// TIA Portal V17 program export: 3 tag tables, 24 data types, 1 data blocks, 11 code blocks (in call order from the OBs), 7 instance data blocks

VAR_GLOBAL   // PLC tag table "Default tag table"
END_VAR

VAR_GLOBAL   // PLC tag table "LPMLV2022_PackTags_Constants"
END_VAR
VAR_GLOBAL CONSTANT   // user constants
   LPMLV2022_COMMAND_PARAMETER_BOOL_UPPER_LIM : UInt := 0;   // Size [0..UPPER_LIM] of structured Array of Unit/Machine Parameter information for values with BOOL data type
   LPMLV2022_COMMAND_PARAMETER_DINT_UPPER_LIM : UInt := 0;   // Size [0..UPPER_LIM] of structured Array of Unit/Machine Parameter information for values with DINT data type
   LPMLV2022_COMMAND_PARAMETER_REAL_UPPER_LIM : UInt := 0;   // Size [0..UPPER_LIM] of structured Array of Unit/Machine Parameter information for values with REAL data type
   LPMLV2022_COMMAND_PARAMETER_LREAL_UPPER_LIM : UInt := 0;   // Size [0..UPPER_LIM] of structured Array of Unit/Machine Parameter information for values with LREAL data type
   LPMLV2022_COMMAND_PARAMETER_STRING_UPPER_LIM : UInt := 0;   // Size [0..UPPER_LIM] of structured Array of Unit/Machine Parameter information for values with STRING data type
   LPMLV2022_COMMAND_RECIPE_UPPER_LIM : UInt := 0;   // Size [0..UPPER_LIM] of structured Array of Recipe Information
   LPMLV2022_COMMAND_PROCESS_VARIABLES_PARAMETER_BOOL_UPPER_LIM : UInt := 0;   // Size [0..UPPER_LIM] of structured Array of Recipe Process Variable information for values with BOOL data type
   LPMLV2022_COMMAND_PROCESS_VARIABLES_PARAMETER_DINT_UPPER_LIM : UInt := 0;   // Size [0..UPPER_LIM] of structured Array of Recipe Process Variable Information for values with DINT data type
   LPMLV2022_COMMAND_PROCESS_VARIABLES_PARAMETER_REAL_UPPER_LIM : UInt := 0;   // Size [0..UPPER_LIM] of structured Array of Recipe Process Variable information for values with REAL data type
   LPMLV2022_COMMAND_PROCESS_VARIABLES_PARAMETER_LREAL_UPPER_LIM : UInt := 0;   // Size [0..UPPER_LIM] of structured Array of Recipe Process Variable information for values with LREAL data type
   LPMLV2022_COMMAND_PROCESS_VARIABLES_PARAMETER_STRING_UPPER_LIM : UInt := 0;   // Size [0..UPPER_LIM] of structured Array of Recipe Process Variable information for values with STRING data type
   LPMLV2022_COMMAND_INGREDIENTS_PARAMETER_BOOL_UPPER_LIM : UInt := 0;   // Size [0..UPPER_LIM] of structured Array of Ingredient information for values with BOOL data type
   LPMLV2022_COMMAND_INGREDIENTS_PARAMETER_DINT_UPPER_LIM : UInt := 0;   // Size [0..UPPER_LIM] of structured Array of Ingredient Information for values with DINT data type
   LPMLV2022_COMMAND_INGREDIENTS_PARAMETER_REAL_UPPER_LIM : UInt := 0;   // Size [0..UPPER_LIM] of structured Array of Ingredient information for values with REAL data type
   LPMLV2022_COMMAND_INGREDIENTS_PARAMETER_LREAL_UPPER_LIM : UInt := 0;   // Size [0..UPPER_LIM] of structured Array of Ingredient information for values with LREAL data type
   LPMLV2022_COMMAND_INGREDIENTS_PARAMETER_STRING_UPPER_LIM : UInt := 0;   // Size [0..UPPER_LIM] of structured Array of Ingredient information for values with STRING data type
   LPMLV2022_STATUS_PARAMETER_BOOL_UPPER_LIM : UInt := 0;   // Size [0..UPPER_LIM] of structured Array of Unit/Machine Parameter information for values with BOOL data type
   LPMLV2022_STATUS_PARAMETER_DINT_UPPER_LIM : UInt := 0;   // Size [0..UPPER_LIM] of structured Array of Unit/Machine Parameter information for values with DINT data type
   LPMLV2022_STATUS_PARAMETER_REAL_UPPER_LIM : UInt := 0;   // Size [0..UPPER_LIM] of structured Array of Unit/Machine Parameter information for values with REAL data type
   LPMLV2022_STATUS_PARAMETER_LREAL_UPPER_LIM : UInt := 0;   // Size [0..UPPER_LIM] of structured Array of Unit/Machine Parameter information for values with LREAL data type
   LPMLV2022_STATUS_PARAMETER_STRING_UPPER_LIM : UInt := 0;   // Size [0..UPPER_LIM] of structured Array of Unit/Machine Parameter information for values with STRING data type
   LPMLV2022_STATUS_RECIPE_UPPER_LIM : UInt := 0;   // Size [0..UPPER_LIM] of structured Array of Recipe Information
   LPMLV2022_STATUS_PROCESS_VARIABLES_PARAMETER_BOOL_UPPER_LIM : UInt := 0;   // Size [0..UPPER_LIM] of structured Array of Recipe Process Variable information for values with BOOL data type
   LPMLV2022_STATUS_PROCESS_VARIABLES_PARAMETER_DINT_UPPER_LIM : UInt := 0;   // Size [0..UPPER_LIM] of structured Array of Recipe Process Variable Information for values with DINT data type
   LPMLV2022_STATUS_PROCESS_VARIABLES_PARAMETER_REAL_UPPER_LIM : UInt := 0;   // Size [0..UPPER_LIM] of structured Array of Recipe Process Variable information for values with REAL data type
   LPMLV2022_STATUS_PROCESS_VARIABLES_PARAMETER_LREAL_UPPER_LIM : UInt := 0;   // Size [0..UPPER_LIM] of structured Array of Recipe Process Variable information for values with LREAL data type
   LPMLV2022_STATUS_PROCESS_VARIABLES_PARAMETER_STRING_UPPER_LIM : UInt := 0;   // Size [0..UPPER_LIM] of structured Array of Recipe Process Variable information for values with STRING data type
   LPMLV2022_STATUS_INGREDIENTS_PARAMETER_BOOL_UPPER_LIM : UInt := 0;   // Size [0..UPPER_LIM] of structured Array of Ingredient information for values with BOOL data type
   LPMLV2022_STATUS_INGREDIENTS_PARAMETER_DINT_UPPER_LIM : UInt := 0;   // Size [0..UPPER_LIM] of structured Array of Ingredient Information for values with DINT data type
   LPMLV2022_STATUS_INGREDIENTS_PARAMETER_REAL_UPPER_LIM : UInt := 0;   // Size [0..UPPER_LIM] of structured Array of Ingredient information for values with REAL data type
   LPMLV2022_STATUS_INGREDIENTS_PARAMETER_LREAL_UPPER_LIM : UInt := 0;   // Size [0..UPPER_LIM] of structured Array of Ingredient information for values with LREAL data type
   LPMLV2022_STATUS_INGREDIENTS_PARAMETER_STRING_UPPER_LIM : UInt := 0;   // Size [0..UPPER_LIM] of structured Array of Ingredient information for values with STRING data type
   LPMLV2022_STATUS_STACK_LIGHT_UPPER_LIM : UInt := 0;   // Size [0..UPPER_LIM] of Indicator for the current stacklight status
   LPMLV2022_ADMIN_PARAMETER_BOOL_UPPER_LIM : UInt := 0;   // Size [0..UPPER_LIM] of structured Array of Unit/Machine Parameter information for values with BOOL data type
   LPMLV2022_ADMIN_PARAMETER_DINT_UPPER_LIM : UInt := 0;   // Size [0..UPPER_LIM] of structured Array of Unit/Machine Parameter information for values with DINT data type
   LPMLV2022_ADMIN_PARAMETER_REAL_UPPER_LIM : UInt := 0;   // Size [0..UPPER_LIM] of structured Array of Unit/Machine Parameter information for values with REAL data type
   LPMLV2022_ADMIN_PARAMETER_LREAL_UPPER_LIM : UInt := 0;   // Size [0..UPPER_LIM] of structured Array of Unit/Machine Parameter information for values with LREAL data type
   LPMLV2022_ADMIN_PARAMETER_STRING_UPPER_LIM : UInt := 0;   // Size [0..UPPER_LIM] of structured Array of Unit/Machine Parameter information for values with STRING data type
   LPMLV2022_ADMIN_ALARM_UPPER_LIM : UInt := 0;   // Size [0..UPPER_LIM] of Array for Machine Alarms
   LPMLV2022_ADMIN_ALARM_HISTORY_UPPER_LIM : UInt := 0;   // Size [0..UPPER_LIM] of Array for Machine Fault Number and Messaging History
   LPMLV2022_ADMIN_WARNING_UPPER_LIM : UInt := 0;   // Size [0..UPPER_LIM] of Machine warnings for general events that do not cause the machine to stop
   LPMLV2022_ADMIN_CUMULATIVE_TIMES_UPPER_LIM : UInt := 0;   // Size [0..UPPER_LIM] of structured Array of Timer Values
   LPMLV2022_ADMIN_NUMBER_OF_MODES_UPPER_LIM : UInt := 8;   // Size [0..UPPER_LIM] of structured Array of Mode and State Time Values for each Cumulative Time Tracker
   LPMLV2022_ADMIN_NUMBER_OF_STATES_UPPER_LIM : UInt := 17;   // Size [0..UPPER_LIM] of state Time Values for each State in each Mode
   LPMLV2022_ADMIN_PRODUCT_DATA_UPPER_LIM : UInt := 0;   // Size [0..UPPER_LIM] of structured array of Product Stream Data
END_VAR

VAR_GLOBAL   // PLC tag table "LPMLV2022_Constants"
END_VAR
VAR_GLOBAL CONSTANT   // user constants
   LPMLV2022_MODE_INVALID : DInt := 0;   // OMAC PackMLV2022 unit mode Invalid
   LPMLV2022_MODE_PRODUCTION : DInt := 1;   // OMAC PackMLV2022 unit mode Production
   LPMLV2022_MODE_MAINTENANCE : DInt := 2;   // OMAC PackMLV2022 unit mode Maintenance
   LPMLV2022_MODE_MANUAL : DInt := 3;   // OMAC PackMLV2022 unit mode Manual
   LPMLV2022_MODE_USER_01 : DInt := 4;   // OMAC PackMLV2022 user-defined unit mode 01
   LPMLV2022_MODE_USER_02 : DInt := 5;   // OMAC PackMLV2022 user-defined unit mode 02
   LPMLV2022_MODE_USER_03 : DInt := 6;   // OMAC PackMLV2022 user-defined unit mode 03
   LPMLV2022_MODE_USER_04 : DInt := 7;   // OMAC PackMLV2022 user-defined unit mode 04
   LPMLV2022_MODE_USER_05 : DInt := 8;   // OMAC PackMLV2022 user-defined unit mode 05
   LPMLV2022_MODE_USER_06 : DInt := 9;   // OMAC PackMLV2022 user-defined unit mode 06
   LPMLV2022_MODE_USER_07 : DInt := 10;   // OMAC PackMLV2022 user-defined unit mode 07
   LPMLV2022_MODE_USER_08 : DInt := 11;   // OMAC PackMLV2022 user-defined unit mode 08
   LPMLV2022_MODE_USER_09 : DInt := 12;   // OMAC PackMLV2022 user-defined unit mode 09
   LPMLV2022_MODE_USER_10 : DInt := 13;   // OMAC PackMLV2022 user-defined unit mode 10
   LPMLV2022_MODE_USER_11 : DInt := 14;   // OMAC PackMLV2022 user-defined unit mode 11
   LPMLV2022_MODE_USER_12 : DInt := 15;   // OMAC PackMLV2022 user-defined unit mode 12
   LPMLV2022_MODE_USER_13 : DInt := 16;   // OMAC PackMLV2022 user-defined unit mode 13
   LPMLV2022_MODE_USER_14 : DInt := 17;   // OMAC PackMLV2022 user-defined unit mode 14
   LPMLV2022_MODE_USER_15 : DInt := 18;   // OMAC PackMLV2022 user-defined unit mode 15
   LPMLV2022_MODE_USER_16 : DInt := 19;   // OMAC PackMLV2022 user-defined unit mode 16
   LPMLV2022_MODE_USER_17 : DInt := 20;   // OMAC PackMLV2022 user-defined unit mode 17
   LPMLV2022_MODE_USER_18 : DInt := 21;   // OMAC PackMLV2022 user-defined unit mode 18
   LPMLV2022_MODE_USER_19 : DInt := 22;   // OMAC PackMLV2022 user-defined unit mode 19
   LPMLV2022_MODE_USER_20 : DInt := 23;   // OMAC PackMLV2022 user-defined unit mode 20
   LPMLV2022_MODE_USER_21 : DInt := 24;   // OMAC PackMLV2022 user-defined unit mode 21
   LPMLV2022_MODE_USER_22 : DInt := 25;   // OMAC PackMLV2022 user-defined unit mode 22
   LPMLV2022_MODE_USER_23 : DInt := 26;   // OMAC PackMLV2022 user-defined unit mode 23
   LPMLV2022_MODE_USER_24 : DInt := 27;   // OMAC PackMLV2022 user-defined unit mode 24
   LPMLV2022_MODE_USER_25 : DInt := 28;   // OMAC PackMLV2022 user-defined unit mode 25
   LPMLV2022_MODE_USER_26 : DInt := 29;   // OMAC PackMLV2022 user-defined unit mode 26
   LPMLV2022_MODE_USER_27 : DInt := 30;   // OMAC PackMLV2022 user-defined unit mode 27
   LPMLV2022_MODE_USER_28 : DInt := 31;   // OMAC PackMLV2022 user-defined unit mode 28
   LPMLV2022_STATE_UNDEFINED : DInt := 0;   // OMAC PackMLV2022 state Undefined
   LPMLV2022_STATE_CLEARING : DInt := 1;   // OMAC PackMLV2022 state Clearing
   LPMLV2022_STATE_STOPPED : DInt := 2;   // OMAC PackMLV2022 state Stopped
   LPMLV2022_STATE_STARTING : DInt := 3;   // OMAC PackMLV2022 state Starting
   LPMLV2022_STATE_IDLE : DInt := 4;   // OMAC PackMLV2022 state Idle
   LPMLV2022_STATE_SUSPENDED : DInt := 5;   // OMAC PackMLV2022 state Suspended
   LPMLV2022_STATE_EXECUTE : DInt := 6;   // OMAC PackMLV2022 state Execute
   LPMLV2022_STATE_STOPPING : DInt := 7;   // OMAC PackMLV2022 state Stopping
   LPMLV2022_STATE_ABORTING : DInt := 8;   // OMAC PackMLV2022 state Aborting
   LPMLV2022_STATE_ABORTED : DInt := 9;   // OMAC PackMLV2022 state Aborted
   LPMLV2022_STATE_HOLDING : DInt := 10;   // OMAC PackMLV2022 state Holding
   LPMLV2022_STATE_HELD : DInt := 11;   // OMAC PackMLV2022 state Held
   LPMLV2022_STATE_UNHOLDING : DInt := 12;   // OMAC PackMLV2022 state Unholding
   LPMLV2022_STATE_SUSPENDING : DInt := 13;   // OMAC PackMLV2022 state Suspending
   LPMLV2022_STATE_UNSUSPENDING : DInt := 14;   // OMAC PackMLV2022 state Unsuspending
   LPMLV2022_STATE_RESETTING : DInt := 15;   // OMAC PackMLV2022 state Resetting
   LPMLV2022_STATE_COMPLETING : DInt := 16;   // OMAC PackMLV2022 state Completing
   LPMLV2022_STATE_COMPLETED : DInt := 17;   // OMAC PackMLV2022 state Completed
   LPMLV2022_CMD_UNDEFINED : DInt := 0;   // OMAC PackMLV2022 control command Undefined
   LPMLV2022_CMD_RESET : DInt := 1;   // OMAC PackMLV2022 control command Reset
   LPMLV2022_CMD_START : DInt := 2;   // OMAC PackMLV2022 control command Start
   LPMLV2022_CMD_STOP : DInt := 3;   // OMAC PackMLV2022 control command Stop
   LPMLV2022_CMD_HOLD : DInt := 4;   // OMAC PackMLV2022 control command Hold
   LPMLV2022_CMD_UNHOLD : DInt := 5;   // OMAC PackMLV2022 control command Unhold
   LPMLV2022_CMD_SUSPEND : DInt := 6;   // OMAC PackMLV2022 control command Suspend
   LPMLV2022_CMD_UNSUSPEND : DInt := 7;   // OMAC PackMLV2022 control command Unsuspend
   LPMLV2022_CMD_ABORT : DInt := 8;   // OMAC PackMLV2022 control command Abort
   LPMLV2022_CMD_CLEAR : DInt := 9;   // OMAC PackMLV2022 control command Clear
   LPMLV2022_CMD_COMPLETE : DInt := 10;   // OMAC PackMLV2022 control command Complete
   LPMLV2022_DIAG_BUFFER_UPPER_LIM : Int := 7;   // Diagnostics buffer array upper boundary (0-based)
   LPMLV2022_MODES_UPPER_LIM : Int := 8;   // (Number of unit modes - 1) -> Array[0..LPMLV2022_MODES_UPPER_LIM]
   LPMLV2022_STATES_UPPER_LIM : Int := 17;   // (Number of states - 1) -> Array[0..LPMLV2022_STATES_UPPER_LIM]
   LPMLV2022_MAX_MODES_UPPER_LIM : Int := 31;   // (Maximum number of unit modes - 1) -> Array[0..LPMLV2022_MAX_MODES_UPPER_LIM]
END_VAR

TYPE "LPMLV2022_typePackTags"
TITLE = LPMLV2022_typePackTags
// Support: tech.team.motioncontrol@siemens.com
// stored: IsFailsafeCompliant false
   STRUCT
      Command : "LPMLV2022_typeCommand";   // Command tags are used to control the operation of the unit/machine. Command tags include unit state commands which control the state transitions in the base state model. The command tags also include parameters and process variables which control how the machine operates
      Status { ExternalWritable := 'False'} : "LPMLV2022_typeStatus";   // Status tags are used to describe the operation of the unit/machine. Status tags include state commands which describe the state transitions in the base state model. The status tags also include parameters and process variables which describe how the machine operates
      Admin { ExternalWritable := 'False'} : "LPMLV2022_typeAdmin";   // Administration tags are used to describe the quality and alarm information of the unit/machine. Administration tags include alarm parameters which describe the conditions within the base state model typically for production data acquisition (PDA) systems. The administration tags also include parameters which can describe how well the machine operates, or specific information on the product quality produced by the machine
   END_STRUCT;
END_TYPE

TYPE "LPMLV2022_typeConfiguration"
TITLE = LPMLV2022_typeConfiguration
// Support: tech.team.motioncontrol@siemens.com
// stored: IsFailsafeCompliant false
   STRUCT
      EnabledModesCfg : DWord := 16#0000_01FE;   // Bit locations within the DWORD represent Mode numbers. A value of 1 in a bit location [0-31] indicates that the corresponding Mode number is enabled. Mode 0 is an Invalid Mode, therefore bit 0 is unused
      DisabledStatesCfg : Array[0.."LPMLV2022_MAX_MODES_UPPER_LIM"] of DWord;   // The array index represents the Mode number. Bit locations within the DWORD value represent State numbers. A value of 1 in a bit location indicates that the corresponding state number is disabled. State 0 is an Undefined State, therefore bit 0 is unused
      ModeTransitionCfg : Array[0.."LPMLV2022_MAX_MODES_UPPER_LIM"] of DWord;   // The array index represents the Mode number. Bit locations within the DWORD value represent State numbers. A value of 1 in a bit location indicates that a mode transition from the corresponding state number is allowed
      holdCmdCfg : DWord := 16#0000_0060;   // Bit locations within the DWORD value represent State numbers. A value of 1 in a bit location indicates that the Hold control command is taken into account in the corresponding state. Note: a state change is only performed if the Holding/Held states are not disabled. The 'holdCmdCfg' can only be activated for the following states: Idle, Starting, Execute, Completing, Completed, Suspending, Suspended, Unsuspending, Unholding
      completeCmdCfg : DWord := 16#0000_0860;   // Bit locations within the DWORD value represent State numbers. A value of 1 in a bit location indicates that the Complete control command is taken into account in the corresponding state. Note: a state change is only performed if the Completing/Completed states are not disabled. The 'completeCmdCfg' can only be activated for the following states: Execute, Suspended, Held
   END_STRUCT;
   // ModeTransitionCfg[1..31] := 16#0000_0214;
END_TYPE

TYPE "LPMLV2022_typeDiagnostics"
TITLE = LPMLV2022_typeDiagnostics
// Support: tech.team.motioncontrol@siemens.com
// stored: IsFailsafeCompliant false
   STRUCT
      bufferIndex { ExternalWritable := 'False'} : Int := -1;   // Index of actual buffer entry
      buffer { ExternalWritable := 'False'} : Array[0.."LPMLV2022_DIAG_BUFFER_UPPER_LIM"] of "LPMLV2022_typeDiagnosticsEntry";   // Diagnostics information buffer
   END_STRUCT;
END_TYPE

TYPE "LPMLV2022_typeDiagnosticsEntry"
TITLE = LPMLV2022_typeDiagnosticsEntry
// Support: tech.team.motioncontrol@siemens.com
// stored: IsFailsafeCompliant false
   STRUCT
      timestamp { ExternalWritable := 'False'} : DTL;   // Timestamp for this entry
      UnitModeCurrent { ExternalWritable := 'False'} : SInt;   // Current unit mode
      StateCurrent { ExternalWritable := 'False'} : SInt;   // Current state
      UnitMode { ExternalWritable := 'False'} : SInt;   // Requested unit mode
      CntrlCmd { ExternalWritable := 'False'} : SInt;   // Request control command
      SC { ExternalWritable := 'False'} : Bool;   // State complete signal
      message { ExternalWritable := 'False'} : Byte;   // Message for this entry
   END_STRUCT;
END_TYPE

TYPE "LPMLV2022_typeAdmin"
TITLE = LPMLV2022_typeAdmin
// Support: tech.team.motioncontrol@siemens.com
// stored: IsFailsafeCompliant false
   STRUCT
      Parameter_REAL { ExternalWritable := 'False'} : Array[0.."LPMLV2022_ADMIN_PARAMETER_REAL_UPPER_LIM"] of "LPMLV2022_typeParameter_REAL";   // Structured Array of Unit/Machine Parameter information for values with REAL data type
      Parameter_STRING { ExternalWritable := 'False'} : Array[0.."LPMLV2022_ADMIN_PARAMETER_STRING_UPPER_LIM"] of "LPMLV2022_typeParameter_STRING";   // Structured Array of Unit/Machine Parameter information for values with STRING data type
      Parameter_LREAL { ExternalWritable := 'False'} : Array[0.."LPMLV2022_ADMIN_PARAMETER_LREAL_UPPER_LIM"] of "LPMLV2022_typeParameter_LREAL";   // Structured Array of Unit/Machine Parameter information for values with LREAL data type
      Parameter_DINT { ExternalWritable := 'False'} : Array[0.."LPMLV2022_ADMIN_PARAMETER_DINT_UPPER_LIM"] of "LPMLV2022_typeParameter_DINT";   // Structured Array of Unit/Machine Parameter information for values with DINT data type
      Parameter_BOOL { ExternalWritable := 'False'} : Array[0.."LPMLV2022_ADMIN_PARAMETER_BOOL_UPPER_LIM"] of "LPMLV2022_typeParameter_BOOL";   // Structured Array of Unit/Machine Parameter information for values with BOOL data type
      Alarm { ExternalWritable := 'False'} : Array[0.."LPMLV2022_ADMIN_ALARM_UPPER_LIM"] of "LPMLV2022_typeEvent";   // Array of Given Size for Machine Alarms. The alarm tags associated to the local interface are typically used as parameters that are displayed or used on the unit locally, for example from an HMI. These alarm parameters can be used to display any alarm, or machine downtime cause that is currently occurring in the system
      AlarmExtent { ExternalWritable := 'False'} : DInt;   // Extent of Alarm Array. The alarm extent is associated with the maximum number of alarms needed for the machine annunciation or reporting
      AlarmHistory { ExternalWritable := 'False'} : Array[0.."LPMLV2022_ADMIN_ALARM_HISTORY_UPPER_LIM"] of "LPMLV2022_typeEvent";   // Array of Given Size for Machine Fault Number and Messaging History. The AlarmHistory array is reserved for alarms that have occurred on the unit/machine and can be sorted in chronological order with the most recently occurring alarmed indexed as Admin.AlarmHistory[0]
      AlarmHistoryExtent { ExternalWritable := 'False'} : DInt;   // Extent of Alarm History Array. The alarm history extent is associated with the maximum number of alarms needed to be archived or tagged as alarm history for the machine
      StopReason { ExternalWritable := 'False'} : "LPMLV2022_typeEvent";   // Machine Stop Reason is typically used for "First Out Fault" Reporting and Other Stoppage Events. The stop reason is the first event captured during an abort, held, suspended or stop event
      Warning { ExternalWritable := 'False'} : Array[0.."LPMLV2022_ADMIN_WARNING_UPPER_LIM"] of "LPMLV2022_typeEvent";   // Machine warnings are for general events that do not cause the machine to stop, but may require operator action as a stoppage may be imminent. Warnings are not typically stored in history
      WarningExtent { ExternalWritable := 'False'} : DInt;   // Extent of Warning Array. The warning extent is associated with the maximum number of warnings needed to be archived or tagged as warnings for the machine
      ModeTimeCurrent { ExternalWritable := 'False'} : DInt;   // Current Mode Time. This tag represents the current amount of time (in seconds) spent in the current Mode as indicated by Status.UnitModeCurrent. The value will start from 0 every time the Mode is changed
      StateTimeCurrent { ExternalWritable := 'False'} : DInt;   // Current State Time. This tag represents the current amount of time (in seconds) spent in the current State as indicated by Status.StateCurrent. The value will start from 0 every time the State is changed
      CumulativeTimes { ExternalWritable := 'False'} : Array[0.."LPMLV2022_ADMIN_CUMULATIVE_TIMES_UPPER_LIM"] of "LPMLV2022_typeCumulativeTimes";   // Structured Array of Timer Values. This tag represents a collection of accumulated time (in seconds) spent in any defined state of any defined mode
      ProductData { ExternalWritable := 'False'} : Array[0.."LPMLV2022_ADMIN_PRODUCT_DATA_UPPER_LIM"] of "LPMLV2022_typeProductData";   // Structured array of Product Stream Data. This tag represents a collection of information about each unique input or output product stream of the machine unit. The extent of the array is typically limited to the maximum number of input and output product streams
      MachDesignSpeed { ExternalWritable := 'False'} : Real;   // Machine Design Speed. This tag represents the maximum design speed of the machine in primary packages per minute for the package configuration being run. This speed is NOT the maximum speed as specified by the manufacturer, but rather the speed of the machine is designed to run in its installed environment
      DisabledStatesCfg { ExternalWritable := 'False'} : Array[0.."LPMLV2022_ADMIN_NUMBER_OF_MODES_UPPER_LIM"] of DWord;   // An array reflecting the Disabled States Configuration for all defined Modes. The array index represents the Mode number. Bit locations within the DWORD value represent State numbers. A value of 1 in a bit location indicates that the corresponding state number is disabled. State 0 is an Undefined State, therefore bit 0 is unused
      CurDisabledStates { ExternalWritable := 'False'} : DWord;   // Reflects the disabled states for the current Mode (Status.UnitModeCurrent). State numbers are represented by bit location. A value of 1 in a certain bit location indicates that the corresponding state number is disabled. State 0 is an Undefined State, therefore bit 0 is unused
      EnabledModesCfg { ExternalWritable := 'False'} : DWord;   // An element reflecting the Enabled Modes Configuration for the unit/machine. Bit locations within the DWORD represent Mode numbers. A value of 1 in a bit location [0-31] indicates that the corresponding Mode number is enabled. Mode 0 is an Invalid Mode, therefore bit 0 is unused
      ModeTransitionCfg { ExternalWritable := 'False'} : Array[0.."LPMLV2022_ADMIN_NUMBER_OF_MODES_UPPER_LIM"] of DWord;   // An array reflecting the Mode Transition Configuration for all modes of the unit/machine. The array index represents the Mode number. Bit locations within the DWORD value represent State numbers. A value of 1 in a bit location indicates that a mode transition from the corresponding state number is allowed
      PLCDateTime { ExternalWritable := 'False'} : "LPMLV2022_typeDateTime";   // Current Date and Time of the Programmable Logic Controller
      PLCDateTimeDTL { ExternalWritable := 'False'} : DTL;   // Current Date and Time (DTL) of the Programmable Logic Controller
   END_STRUCT;
END_TYPE

TYPE "LPMLV2022_typeCommand"
TITLE = LPMLV2022_typeCommand
// Support: tech.team.motioncontrol@siemens.com
// stored: IsFailsafeCompliant false
   STRUCT
      UnitMode : DInt;   // Unit Mode Target (0: Invalid, 1: Production, 2: Maintenance, 3: Manual, 04 - 31: User Definable). Minimum required for supervisory control
      UnitModeChangeRequest : Bool;   // Request Unit Mode Change to Unit Mode Target. Minimum required for supervisory control
      MachSpeed : Real;   // Current Machine Speed Setpoint; Unit of Measure: Primary Packages/Minute. Minimum required for supervisory control
      MaterialInterlock : DWord;   // Materials Ready. It is comprised of a series of bits with 1 equaling ready or not low, 0 equaling not ready, or low. Each bit represents a different user material. Unused bits should be forced to a value of 1 or TRUE
      CntrlCmd : DInt;   // Control Command (0: Undefined, 1: Reset, 2: Start, 3: Stop, 4: Hold, 5: UnHold, 6: Suspend, 7: UnSuspend, 8: Abort, 9: Clear, 10: Complete). Minimum required for supervisory control
      CmdChangeRequest : Bool;   // State Change Request. This CmdChangeRequest bit will command the machine to proceed to change the state to the target state. Minimum required for supervisory control
      Parameter_REAL : Array[0.."LPMLV2022_COMMAND_PARAMETER_REAL_UPPER_LIM"] of "LPMLV2022_typeParameter_REAL";   // Structured Array of Unit/Machine Parameter information for values with REAL data type
      Parameter_STRING : Array[0.."LPMLV2022_COMMAND_PARAMETER_STRING_UPPER_LIM"] of "LPMLV2022_typeParameter_STRING";   // Structured Array of Unit/Machine Parameter information for values with STRING data type
      Parameter_LREAL : Array[0.."LPMLV2022_COMMAND_PARAMETER_LREAL_UPPER_LIM"] of "LPMLV2022_typeParameter_LREAL";   // Structured Array of Unit/Machine Parameter information for values with LREAL data type
      Parameter_DINT : Array[0.."LPMLV2022_COMMAND_PARAMETER_DINT_UPPER_LIM"] of "LPMLV2022_typeParameter_DINT";   // Structured Array of Unit/Machine Parameter information for values with DINT data type
      Parameter_BOOL : Array[0.."LPMLV2022_COMMAND_PARAMETER_BOOL_UPPER_LIM"] of "LPMLV2022_typeParameter_BOOL";   // Structured Array of Unit/Machine Parameter information for values with BOOL data type
      SelectedRecipe : DInt;   // Recipe Selection. This tag is used to designate which recipe should be run on the machine to produce the primary output product, according to a user-design recipe handling procedure. It is designed to correspond directly to the listing in the Recipe Array
      RecipeChangeRequest : Bool;   // Recipe change request. This tag is used to trigger a user-defined recipe changeover process that will configure the machine to produce the primary product designated in Command.SelectedRecipe
      Recipe : Array[0.."LPMLV2022_COMMAND_RECIPE_UPPER_LIM"] of "LPMLV2022_typeCommandRecipe";   // Structured Array of Recipe Information. The recipe data type can be used for defining product ingredient and product processing parameter variables
   END_STRUCT;
END_TYPE

TYPE "LPMLV2022_typeStatus"
TITLE = LPMLV2022_typeStatus
// Support: tech.team.motioncontrol@siemens.com
// stored: IsFailsafeCompliant false
   STRUCT
      UnitModeCurrent { ExternalWritable := 'False'} : DInt;   // Current Unit Mode Number (0: Invalid, 1: Production, 2: Maintenance, 3: Manual, 04 - 31: User Definable). Minimum required for information/machine monitoring
      UnitModeRequested { ExternalWritable := 'False'} : Bool;   // Requested Unit Mode Change. When a unit mode request takes place a numerical value must be present in the unit mode target to change the unit mode
      UnitModeChangeInProcess { ExternalWritable := 'False'} : Bool;   // Requested Unit Mode Change In Process
      StateCurrent { ExternalWritable := 'False'} : DInt;   // Current State Number (0: Undefined, 1: CLEARING, 2: STOPPED, 3: STARTING, 4: IDLE, 5: SUSPENDED, 6: EXECUTE, 7: STOPPING, 8: ABORTING, 9: ABORTED; 10: HOLDING, 11: HELD, 12: UNHOLDING, 13: SUSPENDING, 14: UNSUSPENDING, 15: RESETTING, 16: COMPLETING, 17: COMPLETED). Minimum required for information/machine monitoring
      StateRequested { ExternalWritable := 'False'} : DInt;   // Target State. This value is used for state transition checking, to ensure that transition to a target state can be achieved
      StateChangeInProcess { ExternalWritable := 'False'} : Bool;   // State Change in Process. This bit indicates that a change in state is in progress following a state change request command
      MachSpeed { ExternalWritable := 'False'} : Real;   // Current Machine Speed Setpoint. This describes the set point for the current speed of the machine in primary packages per minute. Minimum required for information/machine monitoring
      CurMachSpeed { ExternalWritable := 'False'} : Real;   // Current Actual Machine Speed. This is the actual value of the machine speed in primary packages per minute. Minimum required for information/machine monitoring
      MaterialInterlock { ExternalWritable := 'False'} : DWord;   // Materials Ready. MaterialInterlock describes the status of the materials that are ready for processing. It is comprised of a series of bits with 1 equaling ready or not low, 0 equaling not ready, or low. Each bit represents a different user material
      EquipmentInterlock { ExternalWritable := 'False'} : "LPMLV2022_typeEquipmentInterlock";   // Is a collection of tags that are used to provide an indicator of Blocked or Starved conditions at the machine unit when integrated into a complete production line
      Parameter_REAL { ExternalWritable := 'False'} : Array[0.."LPMLV2022_STATUS_PARAMETER_REAL_UPPER_LIM"] of "LPMLV2022_typeParameter_REAL";   // Structured Array of Unit/Machine Parameter information for values with REAL data type
      Parameter_STRING { ExternalWritable := 'False'} : Array[0.."LPMLV2022_STATUS_PARAMETER_STRING_UPPER_LIM"] of "LPMLV2022_typeParameter_STRING";   // Structured Array of Unit/Machine Parameter information for values with STRING data type
      Parameter_LREAL { ExternalWritable := 'False'} : Array[0.."LPMLV2022_STATUS_PARAMETER_LREAL_UPPER_LIM"] of "LPMLV2022_typeParameter_LREAL";   // Structured Array of Unit/Machine Parameter information for values with LREAL data type
      Parameter_DINT { ExternalWritable := 'False'} : Array[0.."LPMLV2022_STATUS_PARAMETER_DINT_UPPER_LIM"] of "LPMLV2022_typeParameter_DINT";   // Structured Array of Unit/Machine Parameter information for values with DINT data type
      Parameter_BOOL { ExternalWritable := 'False'} : Array[0.."LPMLV2022_STATUS_PARAMETER_BOOL_UPPER_LIM"] of "LPMLV2022_typeParameter_BOOL";   // Structured Array of Unit/Machine Parameter information for values with BOOL data type
      RecipeCurrent { ExternalWritable := 'False'} : DInt;   // The recipe currently running in production
      RecipeRequested { ExternalWritable := 'False'} : DInt;   // A reflection of the recipe currently selected for production
      RecipeChangeInProcess { ExternalWritable := 'False'} : Bool;   // An indicator for the user-defined recipe changeover process
      Recipe { ExternalWritable := 'False'} : Array[0.."LPMLV2022_STATUS_RECIPE_UPPER_LIM"] of "LPMLV2022_typeStatusRecipe";   // Structured Array of Recipe Information. The recipe data type can be used for defining product ingredient and product processing parameter variables
      Stacklight { ExternalWritable := 'False'} : Array[0.."LPMLV2022_STATUS_STACK_LIGHT_UPPER_LIM"] of DWord;   // Indicator for the current stacklight status. This tag can be used simultaneously for reporting stacklight conditions and as control bits for physical outputs. The status of a light in the stack is associated to a particular bit location within the register (Bit 0: Red Solid, 1: Red Flashing, 2: Amber Solid, 3: Amber Flashing, 4: Blue Solid, 5: Blue Flashing, 6: Green Solid, 7: Green Flashing, 8: Horn Solid, 9: Horn Flashing, 10..31: User-Defined)
   END_STRUCT;
END_TYPE

TYPE "LPMLV2022_typeCommandIngredients"
TITLE = LPMLV2022_typeCommandIngredients
// Support: tech.team.motioncontrol@siemens.com
// stored: IsFailsafeCompliant false
   STRUCT
      Parameter_REAL : Array[0.."LPMLV2022_COMMAND_INGREDIENTS_PARAMETER_REAL_UPPER_LIM"] of "LPMLV2022_typeParameter_REAL";   // Structured Array of Ingredient information for values with REAL data type
      Parameter_STRING : Array[0.."LPMLV2022_COMMAND_INGREDIENTS_PARAMETER_STRING_UPPER_LIM"] of "LPMLV2022_typeParameter_STRING";   // Structured Array of Ingredient information for values with STRING data type
      Parameter_LREAL : Array[0.."LPMLV2022_COMMAND_INGREDIENTS_PARAMETER_LREAL_UPPER_LIM"] of "LPMLV2022_typeParameter_LREAL";   // Structured Array of Ingredient information for values with LREAL data type
      Parameter_DINT : Array[0.."LPMLV2022_COMMAND_INGREDIENTS_PARAMETER_DINT_UPPER_LIM"] of "LPMLV2022_typeParameter_DINT";   // Structured Array of Ingredient Information for values with DINT data type
      Parameter_BOOL : Array[0.."LPMLV2022_COMMAND_INGREDIENTS_PARAMETER_BOOL_UPPER_LIM"] of "LPMLV2022_typeParameter_BOOL";   // Structured Array of Ingredient Information for values with BOOL data type
   END_STRUCT;
END_TYPE

TYPE "LPMLV2022_typeCommandProcessVariables"
TITLE = LPMLV2022_typeCommandProcessVariables
// Support: tech.team.motioncontrol@siemens.com
// stored: IsFailsafeCompliant false
   STRUCT
      Parameter_REAL : Array[0.."LPMLV2022_COMMAND_PROCESS_VARIABLES_PARAMETER_REAL_UPPER_LIM"] of "LPMLV2022_typeParameter_REAL";   // Structured Array of Recipe Process Variable information for values with REAL data type
      Parameter_STRING : Array[0.."LPMLV2022_COMMAND_PROCESS_VARIABLES_PARAMETER_STRING_UPPER_LIM"] of "LPMLV2022_typeParameter_STRING";   // Structured Array of Recipe Process Variable information for values with STRING data type
      Parameter_LREAL : Array[0.."LPMLV2022_COMMAND_PROCESS_VARIABLES_PARAMETER_LREAL_UPPER_LIM"] of "LPMLV2022_typeParameter_LREAL";   // Structured Array of Recipe Process Variable information for values with LREAL data type
      Parameter_DINT : Array[0.."LPMLV2022_COMMAND_PROCESS_VARIABLES_PARAMETER_DINT_UPPER_LIM"] of "LPMLV2022_typeParameter_DINT";   // Structured Array of Recipe Process Variable Information for values with DINT data type
      Parameter_BOOL : Array[0.."LPMLV2022_COMMAND_PROCESS_VARIABLES_PARAMETER_BOOL_UPPER_LIM"] of "LPMLV2022_typeParameter_BOOL";   // Structured Array of Recipe Process Variable Information for values with BOOL data type
   END_STRUCT;
END_TYPE

TYPE "LPMLV2022_typeCommandRecipe"
TITLE = LPMLV2022_typeCommandRecipe
// Support: tech.team.motioncontrol@siemens.com
// stored: IsFailsafeCompliant false
   STRUCT
      ID : DInt;   // ID Value of the Recipe. The ID is used to indicate to the machine which recipe is being produced
      "Name" : String[80];   // Name of Recipe. The Recipe Name is used to further identify the product being produced, especially when alphanumeric characters are used (i.e. SKU or UPC)
      Unit : String[6];   // Unit of Measure of Recipe. The Recipe Unit is used to describe the unit of production for the product being produced
      PrimaryQty : Real;   // Primary Quantity Value of Recipe. PrimaryQty is used to provide a common reference for manufacturing throughput across all the machines on a production line. This element describes the number of Primary Products per recipe Unit for the product being produced by this unit/machine
      ProcessVariables : "LPMLV2022_typeCommandProcessVariables";   // Process Variables for each Recipe. The ProcessVariables structure can be used to hold particular set points needed by the unit/machine for the processing of a specific recipe
      Ingredients : "LPMLV2022_typeCommandIngredients";   // Ingredient Information for each Recipe. The Ingredients structure can be used to hold information for the raw materials that are used by the unit/machine in the processing of a particular product or recipe
   END_STRUCT;
END_TYPE

TYPE "LPMLV2022_typeCumulativeTimes"
TITLE = LPMLV2022_typeCumulativeTimes
// Support: tech.team.motioncontrol@siemens.com
// stored: IsFailsafeCompliant false
   STRUCT
      AccTimeSinceReset { ExternalWritable := 'False'} : DInt;   // Accumulated Time Since Last Reset. The tag represents the amount of time (in seconds) since the reset has been triggered for a particular collection of cumulative times. When a reset for a particular collection is triggered, all times inside the structure for that collection are reset
      ModeStateTimes { ExternalWritable := 'False'} : Array[0.."LPMLV2022_ADMIN_NUMBER_OF_MODES_UPPER_LIM"] of "LPMLV2022_typeModeStateTimes";   // Structured Array of Mode and State Time Values for each Cumulative Time Tracker. This tag is a collection of times for modes and states since the last timer reset was executed
   END_STRUCT;
END_TYPE

TYPE "LPMLV2022_typeDateTime"
TITLE = LPMLV2022_typeDateTime
// Support: tech.team.motioncontrol@siemens.com
// stored: IsFailsafeCompliant false
   STRUCT
      Year { ExternalWritable := 'False'} : Int;
      Month { ExternalWritable := 'False'} : Int;
      Day { ExternalWritable := 'False'} : Int;
      Hour { ExternalWritable := 'False'} : Int;   // (24hr format)
      Minute { ExternalWritable := 'False'} : Int;
      Second { ExternalWritable := 'False'} : Int;
      Millisecond { ExternalWritable := 'False'} : Int;
   END_STRUCT;
END_TYPE

TYPE "LPMLV2022_typeEquipmentInterlock"
TITLE = LPMLV2022_typeEquipmentInterlock
// Support: tech.team.motioncontrol@siemens.com
// stored: IsFailsafeCompliant false
   STRUCT
      Blocked { ExternalWritable := 'False'} : Bool;   // Indicator for Unit/Machine Blocked. This bit, when set to 1, indicates that a downstream system is not able to accept product. In this condition, the equipment is capable of producing product but is in a suspended state due to a downstream system
      Starved { ExternalWritable := 'False'} : Bool;   // Indicator for Unit/Machine Starved. This bit, when set to 1, indicates that an upstream system is not able to supply product. In this condition, the equipment is capable of producing product but is in a suspended state due to an upstream system
   END_STRUCT;
END_TYPE

TYPE "LPMLV2022_typeEvent"
TITLE = LPMLV2022_typeEvent
// Support: tech.team.motioncontrol@siemens.com
// stored: IsFailsafeCompliant false
   STRUCT
      Trigger { ExternalWritable := 'False'} : Bool;   // Alarm Message Trigger. Alarm trigger should be turned on only when the alarm is currently active
      ID { ExternalWritable := 'False'} : DInt;   // Alarm Message Identification Number. The alarm ID number is a unique value assigned to each alarm. Minimum required for information/machine monitoring
      Value { ExternalWritable := 'False'} : DInt;   // Alarm Message Number. The alarm message number is a value that is associated to the alarm allowing for user specific detail or to break down the Alarm.ID to greater detail
      Message { ExternalWritable := 'False'} : String[80];   // Alarm Message. The alarm message is the actual text of the alarm for those machines capable of providing string information
      Category { ExternalWritable := 'False'} : DInt;   // Alarm Category. Alarm category is used to identity what type of alarm has occurred (e.g. electrical, mechanical, materials, utilities, etc.)
      DateTime { ExternalWritable := 'False'} : "LPMLV2022_typeDateTime";   // Date and Time the Alarm Occurred. The timestamp for when the alarm was first triggered
      DateTimeDTL { ExternalWritable := 'False'} : DTL;   // Date and Time (DTL) the Alarm Occurred. The timestamp for when the alarm was first triggered
      AckDateTime { ExternalWritable := 'False'} : "LPMLV2022_typeDateTime";   // Date and Time the Alarm was Acknowledged. The timestamp for when the alarm was acknowledged by the operator, or cleared
      AckDateTimeDTL { ExternalWritable := 'False'} : DTL;   // Date and Time (DTL) the Alarm was Acknowledged. The timestamp for when the alarm was acknowledged by the operator, or cleared
   END_STRUCT;
END_TYPE

TYPE "LPMLV2022_typeModeStateTimes"
TITLE = LPMLV2022_typeModeStateTimes
// Support: tech.team.motioncontrol@siemens.com
// stored: IsFailsafeCompliant false
   STRUCT
      Mode { ExternalWritable := 'False'} : DInt;   // Mode Time Values for each Mode. This tag represents the cumulative amount of time (in seconds) spent in each Mode since the last timer and counter reset was executed
      State { ExternalWritable := 'False'} : Array[0.."LPMLV2022_ADMIN_NUMBER_OF_STATES_UPPER_LIM"] of DInt;   // State Time Values for each State in each Mode. This tag represents the cumulative amount of time (in seconds) spent in each state of a particular Mode since the last timer and counter reset was executed
   END_STRUCT;
END_TYPE

TYPE "LPMLV2022_typeParameter_BOOL"
TITLE = LPMLV2022_typeParameter_BOOL
// Support: tech.team.motioncontrol@siemens.com
// stored: IsFailsafeCompliant false
   STRUCT
      ID : DInt;   // ID Value of Parameter. This is the arbitrary (user defined) ID value of the parameter
      "Name" : String[80];   // Name of Parameter. The literal parameter name is used to describe the parameter number, and its associated value
      Unit : String[6];   // Unit of Measure of Parameter. The parameter unit is typically not used for boolean values
      Value : Bool;   // Value of Parameter. This is the boolean value of the parameter (0: false, 1: true)
   END_STRUCT;
END_TYPE

TYPE "LPMLV2022_typeParameter_DINT"
TITLE = LPMLV2022_typeParameter_DINT
// Support: tech.team.motioncontrol@siemens.com
// stored: IsFailsafeCompliant false
   STRUCT
      ID : DInt;   // ID Value of Parameter. This is the arbitrary (user defined) ID value of the parameter
      "Name" : String[80];   // Name of Parameter. The literal parameter name is used to describe the parameter number, and its associated value
      Unit : String[6];   // Unit of Measure of Parameter. An example parameter unit of measure may be DegF, secs, PPM, revs, mm, etc.
      Value : DInt;   // Value of Parameter. This is the numeric value of the parameter
   END_STRUCT;
END_TYPE

TYPE "LPMLV2022_typeParameter_LREAL"
TITLE = LPMLV2022_typeParameter_LREAL
// Support: tech.team.motioncontrol@siemens.com
// stored: IsFailsafeCompliant false
   STRUCT
      ID : DInt;   // ID Value of Parameter. This is the arbitrary (user defined) ID value of the parameter
      "Name" : String[80];   // Name of Parameter. The literal parameter name is used to describe the parameter number, and its associated value
      Unit : String[6];   // Unit of Measure of Parameter. An example parameter unit of measure may be DegF, secs, PPM, revs, mm, etc.
      Value : LReal;   // Value of Parameter. This is the numeric value of the parameter
   END_STRUCT;
END_TYPE

TYPE "LPMLV2022_typeParameter_REAL"
TITLE = LPMLV2022_typeParameter_REAL
// Support: tech.team.motioncontrol@siemens.com
// stored: IsFailsafeCompliant false
   STRUCT
      ID : DInt;   // ID Value of Parameter. This is the arbitrary (user defined) ID value of the parameter
      "Name" : String[80];   // Name of Parameter. The literal parameter name is used to describe the parameter number, and its associated value
      Unit : String[6];   // Unit of Measure of Parameter. An example parameter unit of measure may be DegF, secs, PPM, revs, mm, etc.
      Value : Real;   // Value of Parameter. This is the numeric value of the parameter
   END_STRUCT;
END_TYPE

TYPE "LPMLV2022_typeParameter_STRING"
TITLE = LPMLV2022_typeParameter_STRING
// Support: tech.team.motioncontrol@siemens.com
// stored: IsFailsafeCompliant false
   STRUCT
      ID : DInt;   // ID Value of Parameter. This is the arbitrary (user defined) ID value of the parameter
      "Name" : String[80];   // Name of Parameter. The literal parameter name is used to describe the parameter number, and its associated value
      Unit : String[6];   // Unit of Measure of Parameter. The parameter unit is typically not used for string values
      Value : String[80];   // Value of Parameter. This is the string value of the parameter
   END_STRUCT;
END_TYPE

TYPE "LPMLV2022_typeProductData"
TITLE = LPMLV2022_typeProductData
// Support: tech.team.motioncontrol@siemens.com
// stored: IsFailsafeCompliant false
   STRUCT
      ID { ExternalWritable := 'False'} : DInt;   // ID Number for each Product Stream. The product IDs are used to report product identity for each product stream
      "Name" { ExternalWritable := 'False'} : String[80];   // Name of Product Stream. The Name element is used to further report the identity of the product within the product stream, especially when alphanumeric characters are used (i.e. SKU or UPC)
      Unit { ExternalWritable := 'False'} : String[6];   // Unit of Measure of each Product Stream. The Unit element is used to report the unit of production for the product within the product stream. An example product unit of measure may be Pc, Crtn, Case, etc
      PrimaryQty { ExternalWritable := 'False'} : Real;   // Product Primary Quantity Value of each Product Stream. The PrimaryQty element is used to provide a common reference for manufacturing throughput across all the machines on a production line. This element relates the number of Primary Products per Unit for a particular product stream. It can be used as a conversion factor for a local machine reference speed since Command.MachSpeed is given in units of PrimaryProducts/Min
      ConsumedCount { ExternalWritable := 'False'} : DInt;   // Consumed Count of each Product Stream. This tag represents the material used/consumed in the production machine for a particular input or output product stream. An example of tag usage would be the number of bags consumed in a filler, or bagger packaging machine, or the amount of linear length used, or the number caps used
      ProcessedCount { ExternalWritable := 'False'} : DInt;   // Processed Count of each Product Stream. This tag represents the number of products from a particular input or output product stream processed by the production machine. An example of tag usage would be the number of products that were made, including all good and defective products. The number of products processed minus the number of defective products is the number of products actually made by the machine. Minimum required for information/machine monitoring
      DefectiveCount { ExternalWritable := 'False'} : DInt;   // Defective Count of each Product Stream. This tag represents the number of products from a particular input or output product stream that is marked as defective in the production machine, to be used if applicable. An example of tag usage would be the number of products rejected or products that are termed defective. Minimum required for information/machine monitoring
      AccConsumedCount { ExternalWritable := 'False'} : DInt;   // Accumulated Consumption Count of each Product Stream Consumption Since Last Reset. This tag represents the total accumulated material used/consumed in the production machine for a particular input or output product stream
      AccProcessedCount { ExternalWritable := 'False'} : DInt;   // Accumulated Processed Count of each Product Stream Since Last Reset. This tag represents the total accumulated number of products from a particular input or output product stream processed by the production machine. An example of tag usage would be the number of products that were made, including all good and defective products. The number of products processed minus the number of defective products is the number of products actually made by the machine
      AccDefectiveCount { ExternalWritable := 'False'} : DInt;   // Accumulated Defective Count of each Product Stream Since Last Reset. This tag represents the total accumulated number of products from a particular input or output product stream that is marked as defective in the production machine, to be used if applicable. An example of tag usage would be the number of products rejected or products that are termed defective
   END_STRUCT;
END_TYPE

TYPE "LPMLV2022_typeStatusIngredients"
TITLE = LPMLV2022_typeStatusIngredients
// Support: tech.team.motioncontrol@siemens.com
// stored: IsFailsafeCompliant false
   STRUCT
      Parameter_REAL { ExternalWritable := 'False'} : Array[0.."LPMLV2022_STATUS_INGREDIENTS_PARAMETER_REAL_UPPER_LIM"] of "LPMLV2022_typeParameter_REAL";   // Structured Array of Ingredient information for values with REAL data type
      Parameter_STRING { ExternalWritable := 'False'} : Array[0.."LPMLV2022_STATUS_INGREDIENTS_PARAMETER_STRING_UPPER_LIM"] of "LPMLV2022_typeParameter_STRING";   // Structured Array of Ingredient information for values with STRING data type
      Parameter_LREAL { ExternalWritable := 'False'} : Array[0.."LPMLV2022_STATUS_INGREDIENTS_PARAMETER_LREAL_UPPER_LIM"] of "LPMLV2022_typeParameter_LREAL";   // Structured Array of Ingredient information for values with LREAL data type
      Parameter_DINT { ExternalWritable := 'False'} : Array[0.."LPMLV2022_STATUS_INGREDIENTS_PARAMETER_DINT_UPPER_LIM"] of "LPMLV2022_typeParameter_DINT";   // Structured Array of Ingredient Information for values with DINT data type
      Parameter_BOOL { ExternalWritable := 'False'} : Array[0.."LPMLV2022_STATUS_INGREDIENTS_PARAMETER_BOOL_UPPER_LIM"] of "LPMLV2022_typeParameter_BOOL";   // Structured Array of Ingredient Information for values with BOOL data type
   END_STRUCT;
END_TYPE

TYPE "LPMLV2022_typeStatusProcessVariables"
TITLE = LPMLV2022_typeStatusProcessVariables
// Support: tech.team.motioncontrol@siemens.com
// stored: IsFailsafeCompliant false
   STRUCT
      Parameter_REAL { ExternalWritable := 'False'} : Array[0.."LPMLV2022_STATUS_PROCESS_VARIABLES_PARAMETER_REAL_UPPER_LIM"] of "LPMLV2022_typeParameter_REAL";   // Structured Array of Recipe Process Variable information for values with REAL data type
      Parameter_STRING { ExternalWritable := 'False'} : Array[0.."LPMLV2022_STATUS_PROCESS_VARIABLES_PARAMETER_STRING_UPPER_LIM"] of "LPMLV2022_typeParameter_STRING";   // Structured Array of Recipe Process Variable information for values with STRING data type
      Parameter_LREAL { ExternalWritable := 'False'} : Array[0.."LPMLV2022_STATUS_PROCESS_VARIABLES_PARAMETER_LREAL_UPPER_LIM"] of "LPMLV2022_typeParameter_LREAL";   // Structured Array of Recipe Process Variable information for values with LREAL data type
      Parameter_DINT { ExternalWritable := 'False'} : Array[0.."LPMLV2022_STATUS_PROCESS_VARIABLES_PARAMETER_DINT_UPPER_LIM"] of "LPMLV2022_typeParameter_DINT";   // Structured Array of Recipe Process Variable Information for values with DINT data type
      Parameter_BOOL { ExternalWritable := 'False'} : Array[0.."LPMLV2022_STATUS_PROCESS_VARIABLES_PARAMETER_BOOL_UPPER_LIM"] of "LPMLV2022_typeParameter_BOOL";   // Structured Array of Recipe Process Variable Information for values with BOOL data type
   END_STRUCT;
END_TYPE

TYPE "LPMLV2022_typeStatusRecipe"
TITLE = LPMLV2022_typeStatusRecipe
// Support: tech.team.motioncontrol@siemens.com
// stored: IsFailsafeCompliant false
   STRUCT
      ID { ExternalWritable := 'False'} : DInt;   // ID Value of the Recipe. The ID is used to indicate to the machine which recipe is being produced
      "Name" { ExternalWritable := 'False'} : String[80];   // Name of Recipe. The Recipe Name is used to further identify the product being produced, especially when alphanumeric characters are used (i.e. SKU or UPC)
      Unit { ExternalWritable := 'False'} : String[6];   // Unit of Measure of Recipe. The Recipe Unit is used to describe the unit of production for the product being produced
      PrimaryQty { ExternalWritable := 'False'} : Real;   // Primary Quantity Value of Recipe. PrimaryQty is used to provide a common reference for manufacturing throughput across all the machines on a production line. This element describes the number of Primary Products per recipe Unit for the product being produced by this unit/machine
      ProcessVariables { ExternalWritable := 'False'} : "LPMLV2022_typeStatusProcessVariables";   // Process Variables for each Recipe. The ProcessVariables structure can be used to reflect and confirm particular set points needed by the unit/machine for the processing of a specific recipe or to report production statistics
      Ingredients { ExternalWritable := 'False'} : "LPMLV2022_typeStatusIngredients";   // Ingredient Information for each Recipe. The Ingredients structure can be used to hold information for the raw materials that are used by the unit/machine in the processing of a particular product or recipe. Each element in one of the parameter arrays is considered to be an ingredient
   END_STRUCT;
END_TYPE

DATA_BLOCK "UnitModeStateManagerDiagnosticsForHMI"   // DB30134
{ S7_Optimized_Access := 'TRUE'; DB_Accessible_From_OPC_UA := 'FALSE' }
VERSION : 0.1
// stored: AutoNumber true, DBAccessibleFromOPCUA false, DBAccessibleFromWebserver false, IsOnlyStoredInLoadMemory false, IsRetainMemResEnabled false, IsWriteProtectedInAS false, MemoryReserve 0
   VAR
      actualDiagnosticsBufferIndex { ExternalWritable := 'False'} : Int;   // Index of the actual diagnostics buffer entry of the LPMLV2022_UnitModeStateManager (InstLPMLV2022_UnitModeStateManager.diagnostics.bufferIndex)
      diagnosticsBufferIndexForHMI : Int;   // Index for selecting the diagnostics buffer entry to be displayed on the HMI
      diagnosticsBufferEntryForHMI { ExternalWritable := 'False'} : "LPMLV2022_typeDiagnosticsEntry";   // Selected diagnostics buffer entry (InstLPMLV2022_UnitModeStateManager.diagnostics.buffer[diagnosticsBufferIndexForHMI])
      messageCurrentPLCIndex { ExternalWritable := 'False'} : Byte;   // Message of the actual diagnostics buffer entry of the LPMLV2022_UnitModeStateManager
   END_VAR
BEGIN
END_DATA_BLOCK

ORGANIZATION_BLOCK "Main"   // OB1, LAD, ProgramCycle
TITLE = "Main Program Sweep (Cycle)"
{ S7_Optimized_Access := 'TRUE' }
VERSION : 0.1
// stored: AutoNumber true, IsIECCheckEnabled false, SetENOAutomatically false
   VAR_INPUT
      Initial_Call : Bool;   // Initial call of this OB
      Remanence : Bool;   // =True, if remanent data are available
   END_VAR
BEGIN

REGION Network 1: Example of calling LPMLV2022_UnitModeStateManager incl. ToDo structure
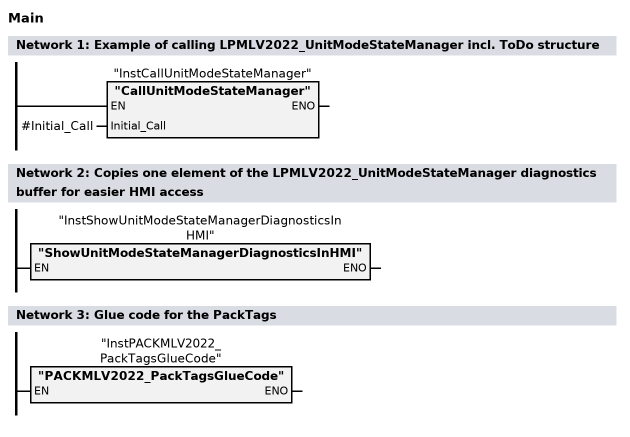
   RUNG wire#powerrail
      "InstCallUnitModeStateManager"(Initial_Call := #Initial_Call)
   END_RUNG
   // the same network as SCL:
   "InstCallUnitModeStateManager"(Initial_Call := #Initial_Call);   // "CallUnitModeStateManager"
END_REGION

REGION Network 2: Copies one element of the LPMLV2022_UnitModeStateManager diagnostics buffer for easier HMI access
   RUNG wire#powerrail
      "InstShowUnitModeStateManagerDiagnosticsInHMI"()
   END_RUNG
   // the same network as SCL:
   "InstShowUnitModeStateManagerDiagnosticsInHMI"();   // "ShowUnitModeStateManagerDiagnosticsInHMI"
END_REGION

REGION Network 3: Glue code for the PackTags
   RUNG wire#powerrail
      "InstPACKMLV2022_PackTagsGlueCode"()
   END_RUNG
   // the same network as SCL:
   "InstPACKMLV2022_PackTagsGlueCode"();   // "PACKMLV2022_PackTagsGlueCode"
END_REGION
END_ORGANIZATION_BLOCK

FUNCTION_BLOCK "CallUnitModeStateManager"
{ S7_Optimized_Access := 'TRUE' }
VERSION : 0.1
   VAR_INPUT 
      Initial_Call { ExternalAccessible := 'False'; ExternalVisible := 'False'; ExternalWritable := 'False'} : Bool;   // Initial call flag from the calling OB
   END_VAR


BEGIN
	REGION HEADER
	  //================================================================================
	  // SIEMENS AG
	  // (c)Copyright 2023 All Rights Reserved
	  //--------------------------------------------------------------------------------
	  // Library: -
	  // Tested with: S7-1513-1 PN with FW version V2.9
	  // Engineering: TIA Portal V17 Update 4
	  // Restrictions: -
	  // Requirements: LPMLV2022
	  // Functionality: Example of calling LPMLV2022_UnitModeStateManager incl. ToDo structure
	  // Support: tech.team.motioncontrol@siemens.com
	  // Note: Parameter comments are only available in language 'English (United States)'
	  //--------------------------------------------------------------------------------
	  // Change log table:
	  // Version  Date        Expert in charge  Changes applied
	  // 01.00.00 28.02.2023  KT                First released version
	  //================================================================================
	END_REGION
	
	// Disable unit modes and set state configuration in modes - default: Base state model
	IF #Initial_Call THEN
	  
	  // Enable the needed unit modes
	  "LPMLV2022_ConfigureEnabledModesCfg"(ProductionMode := TRUE,
	                                       MaintenanceMode := TRUE,
	                                       UserMode01 := TRUE,
	                                       UserMode02 := FALSE,
	                                       UserMode03 := FALSE,
	                                       UserMode04 := FALSE,
	                                       UserMode05 := FALSE,
	                                       UserMode06 := FALSE,
	                                       UserMode07 := FALSE,
	                                       UserMode08 := FALSE,
	                                       UserMode09 := FALSE,
	                                       UserMode10 := FALSE,
	                                       UserMode11 := FALSE,
	                                       UserMode12 := FALSE,
	                                       UserMode13 := FALSE,
	                                       UserMode14 := FALSE,
	                                       UserMode15 := FALSE,
	                                       UserMode16 := FALSE,
	                                       UserMode17 := FALSE,
	                                       UserMode18 := FALSE,
	                                       UserMode19 := FALSE,
	                                       UserMode20 := FALSE,
	                                       UserMode21 := FALSE,
	                                       UserMode22 := FALSE,
	                                       UserMode23 := FALSE,
	                                       UserMode24 := FALSE,
	                                       UserMode25 := FALSE,
	                                       UserMode26 := FALSE,
	                                       UserMode27 := FALSE,
	                                       UserMode28 := FALSE,
	                                       EnabledModesCfg => "InstLPMLV2022_UnitModeStateManager".configuration.EnabledModesCfg);
	  
	  // Set state configuration for every unit mode
	  // Mode: Production
	  "LPMLV2022_ConfigureDisabledStatesCfg"(Clearing := FALSE,
	                                         Starting := FALSE,
	                                         Suspended := FALSE,
	                                         Stopping := FALSE,
	                                         Aborting := FALSE,
	                                         Holding := FALSE,
	                                         Held := FALSE,
	                                         Unholding := FALSE,
	                                         Suspending := FALSE,
	                                         Unsuspending := FALSE,
	                                         Resetting := FALSE,
	                                         Completing := FALSE,
	                                         Completed := FALSE,
	                                         DisabledStatesCfg => "InstLPMLV2022_UnitModeStateManager".configuration.DisabledStatesCfg["LPMLV2022_MODE_PRODUCTION"]);
	  
	  // Mode: Maintenance
	  "LPMLV2022_ConfigureDisabledStatesCfg"(Clearing := FALSE,
	                                         Starting := FALSE,
	                                         Suspended := TRUE,
	                                         Stopping := FALSE,
	                                         Aborting := FALSE,
	                                         Holding := FALSE,
	                                         Held := FALSE,
	                                         Unholding := FALSE,
	                                         Suspending := TRUE,
	                                         Unsuspending := TRUE,
	                                         Resetting := FALSE,
	                                         Completing := FALSE,
	                                         Completed := FALSE,
	                                         DisabledStatesCfg => "InstLPMLV2022_UnitModeStateManager".configuration.DisabledStatesCfg["LPMLV2022_MODE_MAINTENANCE"]);
	  
	  // Mode: Manual
	  "LPMLV2022_ConfigureDisabledStatesCfg"(Clearing := FALSE,
	                                         Starting := FALSE,
	                                         Suspended := TRUE,
	                                         Stopping := FALSE,
	                                         Aborting := FALSE,
	                                         Holding := TRUE,
	                                         Held := TRUE,
	                                         Unholding := TRUE,
	                                         Suspending := TRUE,
	                                         Unsuspending := TRUE,
	                                         Resetting := FALSE,
	                                         Completing := TRUE,
	                                         Completed := TRUE,
	                                         DisabledStatesCfg => "InstLPMLV2022_UnitModeStateManager".configuration.DisabledStatesCfg["LPMLV2022_MODE_MANUAL"]);
	  
	  // Mode: UserMode01
	  "LPMLV2022_ConfigureDisabledStatesCfg"(Clearing := FALSE,
	                                         Starting := FALSE,
	                                         Suspended := TRUE,
	                                         Stopping := FALSE,
	                                         Aborting := FALSE,
	                                         Holding := FALSE,
	                                         Held := FALSE,
	                                         Unholding := FALSE,
	                                         Suspending := TRUE,
	                                         Unsuspending := TRUE,
	                                         Resetting := FALSE,
	                                         Completing := FALSE,
	                                         Completed := FALSE,
	                                         DisabledStatesCfg => "InstLPMLV2022_UnitModeStateManager".configuration.DisabledStatesCfg["LPMLV2022_MODE_USER_01"]);
	  
	  // Mode: UserMode02
	  // "LPMLV2022_ConfigureDisabledStatesCfg"(Clearing := FALSE,
	  //                                        Starting := FALSE,
	  //                                        Suspended := FALSE,
	  //                                        Stopping := FALSE,
	  //                                        Aborting := FALSE,
	  //                                        Holding := FALSE,
	  //                                        Held := FALSE,
	  //                                        Unholding := FALSE,
	  //                                        Suspending := FALSE,
	  //                                        Unsuspending := FALSE,
	  //                                        Resetting := FALSE,
	  //                                        Completing := FALSE,
	  //                                        Completed := FALSE,
	  //                                        DisabledStatesCfg => "InstLPMLV2022_UnitModeStateManager".configuration.DisabledStatesCfg["LPMLV2022_MODE_USER_02"]);
	  
	  RETURN; // Nothing else in this cycle to avoid runtime peaks
	END_IF;
	
	// Call of LPMLV2022_UnitModeStateManager
	// Note: the inputs UnitMode, CntrlCmd, ... are set via the PackTags command tags (see FB PACKMLV2022_PackTagsGlueCode)
	//       the input SC is normally set in the program when the action of an acting state is done, for testing purposes it can be set in the example HMI
	"InstLPMLV2022_UnitModeStateManager"();
	
	// Reset the state complete signal (SC)
	"InstLPMLV2022_UnitModeStateManager".SC := FALSE;
	
	// Functional implementation for all unit modes and states
	CASE "InstLPMLV2022_UnitModeStateManager".UnitModeCurrent OF
	  "LPMLV2022_MODE_PRODUCTION":
	    CASE "InstLPMLV2022_UnitModeStateManager".StateCurrent OF
	      "LPMLV2022_STATE_RESETTING":
	        //-------------------------------------------
	        // State Type: Acting
	        // This state is the result of a Reset command from the Stopped or
	        // Completed state. Faults and stop causes are reset. Resetting will
	        // typically cause safety devices to be energized and place the machine in
	        // the Idle state where it will wait for a Start command. No hazardous
	        // motion should happen in this state.
	        //-------------------------------------------
	        ; // todo
	        
	        // "InstLPMLV2022_UnitModeStateManager".SC := TRUE; // Set state complete signal when action is done
	        
	      "LPMLV2022_STATE_IDLE":
	        //-------------------------------------------
	        // State Type: Wait
	        // This is the state that indicates that Resetting is complete.
	        // The machine will maintain the conditions that were achieved
	        // during the Resetting state, and perform operations required when the
	        // machine is in Idle.
	        //-------------------------------------------
	        ; // todo
	        
	      "LPMLV2022_STATE_STARTING":
	        //-------------------------------------------
	        // State Type: Acting
	        // The machine completes the steps needed to start. This state is entered
	        // as a result of a Start command (local or remote). When Starting completes,
	        // the machine will transition to the Execute state.
	        //-------------------------------------------
	        ; // todo
	        
	        // "InstLPMLV2022_UnitModeStateManager".SC := TRUE; // Set state complete signal when action is done
	        
	      "LPMLV2022_STATE_EXECUTE":
	        //-------------------------------------------
	        // State Type: Acting
	        // Once the machine is processing materials it is in the Execute state
	        // until a transition command is received. Different machine modes
	        // will result in specific types of Execute activities.
	        // For example, if the machine is in the “Production” mode, the Execute will
	        // result in products being produced, while perhaps in a user-defined “Clean Out” mode
	        // the Execute state would result in the action of cleaning the machine.
	        //-------------------------------------------
	        ; // todo
	        
	      "LPMLV2022_STATE_STOPPING":
	        //-------------------------------------------
	        // State Type: Acting
	        // This state is entered in response to a Stop command.
	        // While in this state the machine executes the logic that brings it to a
	        // controlled stop as reflected by the Stopped state. Normal Starting
	        // of the machine cannot be initiated unless Resetting has taken place.
	        //-------------------------------------------
	        ; // todo
	        
	        // "InstLPMLV2022_UnitModeStateManager".SC := TRUE; // Set state complete signal when action is done
	        
	      "LPMLV2022_STATE_STOPPED":
	        //-------------------------------------------
	        // State Type: Wait
	        // The machine is powered and stationary after completing the Stopping state.
	        // All communications with other systems are functioning (if applicable).
	        // A Reset command will cause a transition from Stopped to the Resetting state.
	        //-------------------------------------------
	        ; // todo
	        
	      "LPMLV2022_STATE_HOLDING":
	        //-------------------------------------------
	        // State Type: Acting
	        // This state is used when internal (inside this unit/machine and
	        // not from another machine on the production line) machine conditions do
	        // not allow the machine to continue producing, that is, the machine leaves
	        // the Execute or Suspended states due to internal conditions.
	        // This is typically used for routine machine conditions that require minor
	        // operator servicing to continue production. This state can be initiated
	        // automatically or by an operator and can be easily recovered from.
	        // An example of this would be a machine that requires an operator to
	        // periodically refill a glue dispenser or carton magazine and due to the
	        // machine design, these operations cannot be performed while the machine
	        // is running. Since these types of tasks are normal production operations,
	        // it is not desirable to go through aborting or stopping sequences, and
	        // because these functions are integral to the machine they are not
	        // considered to be “external”. While in the Holding state, the machine is
	        // typically brought to a controlled stop and then transitions to Held upon
	        // state complete. To be able to restart production correctly after the
	        // Held state, all relevant process set points and return status of the
	        // procedures at the time of receiving the Hold command must be saved in
	        // the machine controller when executing the Holding procedure.
	        //-------------------------------------------
	        ; // todo
	        
	        // "InstLPMLV2022_UnitModeStateManager".SC := TRUE; // Set state complete signal when action is done            
	        
	      "LPMLV2022_STATE_HELD":
	        //-------------------------------------------
	        // State Type: Wait
	        // Refer to Holding for when this state is used. In this state the machine
	        // does not produce product. It will either stop running or continue to dry
	        // cycle. A transition to the Unholding state will occur when internal
	        // machine conditions change or an Unhold command is initiated by an operator.
	        //-------------------------------------------
	        ; // todo
	        
	      "LPMLV2022_STATE_UNHOLDING":
	        //-------------------------------------------
	        // State Type: Acting
	        // Refer to Holding for when this state is used. A machine will typically
	        // enter into Unholding automatically when internal conditions,
	        // material levels, for example, return to an acceptable level. If an operator
	        // is required to perform minor servicing to replenish materials or make
	        // adjustments, then the Unhold command may be initiated by the operator.
	        //-------------------------------------------
	        ; // todo
	        
	        // "InstLPMLV2022_UnitModeStateManager".SC := TRUE; // Set state complete signal when action is done   
	        
	      "LPMLV2022_STATE_SUSPENDING":
	        //-------------------------------------------
	        // State Type: Acting
	        // This state is used when external (outside this unit/machine but
	        // usually on the same integrated production line) process conditions do not
	        // allow the machine to continue producing, that is, the machine leaves
	        // Execute due to upstream or downstream conditions on the line. This is
	        // typically due to a Blocked or Starved event. This condition may be
	        // detected by a local machine sensor or based on a supervisory system
	        // external command. While in the Suspending state, the machine is
	        // typically brought to a controlled stop and then transitions to
	        // Suspended upon state complete. To be able to restart production
	        // correctly after the Suspended state, all relevant process set points and
	        // return status of the procedures at the time of receiving the Suspend
	        // command must be saved in the machine controller when executing the
	        // Suspending procedure.
	        //-------------------------------------------
	        ; // todo
	        
	        // "InstLPMLV2022_UnitModeStateManager".SC := TRUE; // Set state complete signal when action is done
	        
	      "LPMLV2022_STATE_SUSPENDED":
	        //-------------------------------------------
	        // State Type: Wait
	        // Refer to Suspending for when this state is used. In this state the
	        // machine does produce product. It will either stop running or continue
	        // to cycle without producing until external process conditions return to
	        // normal, at which time, the Suspended state will transition to the
	        // Unsuspending state, typically without any operator intervention.
	        //-------------------------------------------
	        ; // todo
	        
	      "LPMLV2022_STATE_UNSUSPENDING":
	        //-------------------------------------------
	        // State Type: Acting
	        // Refer to Suspending for when this state is used. This state is a result
	        // of process conditions returning to normal. The Unsuspending state
	        // initiates any required actions or sequences necessary to transition the
	        // machine from Suspended back to Execute. To be able to restart
	        // production correctly after the Suspended state, all relevant process
	        // set points and return status of the procedures at the time of receiving the
	        // Suspend command must be saved in the machine controller when
	        // executing the Suspending procedure.
	        //-------------------------------------------
	        ; // todo
	        
	        // "InstLPMLV2022_UnitModeStateManager".SC := TRUE; // Set state complete signal when action is done
	        
	      "LPMLV2022_STATE_COMPLETING":
	        //-------------------------------------------
	        // State Type: Acting
	        // This state is the result of a Complete command from the Execute, Held
	        // or Suspended states. The Complete command may be internally generated,
	        // such as reaching the end of a predefined production count where normal
	        // operation has run to completion, or externally generated, such as by a
	        // supervisory system. The Completing state is often used to end a
	        // production run and summarize production data.
	        //-------------------------------------------
	        ; // todo
	        
	        // "InstLPMLV2022_UnitModeStateManager".SC := TRUE; // Set state complete signal when action is done
	        
	      "LPMLV2022_STATE_COMPLETED":
	        //-------------------------------------------
	        // State Type: Wait
	        // The machine has finished the Completing state and is now waiting for
	        // a Reset command before transitioning to the Resetting state.
	        //-------------------------------------------
	        ; // todo
	        
	      "LPMLV2022_STATE_ABORTING":
	        //-------------------------------------------
	        // State type: Acting
	        // The Aborting state can be entered at any time in response to the Abort command,
	        // typically triggered by the occurrence of a machine event that warrants an aborting action.
	        // The aborting logic will bring the machine to a rapid safe stop.
	        //-------------------------------------------
	        ; // todo
	        
	        // "InstLPMLV2022_UnitModeStateManager".SC := TRUE; // Set state complete signal when action is done
	        
	      "LPMLV2022_STATE_ABORTED":
	        //-------------------------------------------
	        // State Type: Wait
	        // The machine maintains status information relevant to the abort condition.
	        // The machine can only exit the Aborted state after an explicit Clear command,
	        // subsequent to manual intervention to correct and reset the
	        // detected machine faults.
	        //-------------------------------------------
	        ; // todo
	        
	      "LPMLV2022_STATE_CLEARING":
	        //------------------------------------------
	        // State Type: Acting
	        // Initiated by a Clear command to clear faults that may have occurred and
	        // are present in the Aborted state before proceeding to a Stopped state.
	        //-------------------------------------------
	        ; // todo
	        
	        // "InstLPMLV2022_UnitModeStateManager".SC := TRUE; // Set state complete signal when action is done
	        
	      ELSE
	        // Error reaction
	        ; // todo
	    END_CASE;
	    
	  "LPMLV2022_MODE_MAINTENANCE":
	    CASE "InstLPMLV2022_UnitModeStateManager".StateCurrent OF
	      "LPMLV2022_STATE_RESETTING":
	        ; // todo
	        
	        // "InstLPMLV2022_UnitModeStateManager".SC := TRUE; // Set state complete signal when action is done
	        
	      "LPMLV2022_STATE_IDLE":
	        ; // todo
	        
	      "LPMLV2022_STATE_STARTING":
	        ; // todo
	        
	        // "InstLPMLV2022_UnitModeStateManager".SC := TRUE; // Set state complete signal when action is done
	        
	      "LPMLV2022_STATE_EXECUTE":
	        ; // todo
	        
	      "LPMLV2022_STATE_STOPPING":
	        ; // todo
	        
	        // "InstLPMLV2022_UnitModeStateManager".SC := TRUE; // Set state complete signal when action is done
	        
	      "LPMLV2022_STATE_STOPPED":
	        ; // todo
	        
	      "LPMLV2022_STATE_HOLDING":
	        ; // todo
	        
	        // "InstLPMLV2022_UnitModeStateManager".SC := TRUE; // Set state complete signal when action is done            
	        
	      "LPMLV2022_STATE_HELD":
	        ; // todo
	        
	      "LPMLV2022_STATE_UNHOLDING":
	        ; // todo
	        
	        // "InstLPMLV2022_UnitModeStateManager".SC := TRUE; // Set state complete signal when action is done   
	        
	      "LPMLV2022_STATE_SUSPENDING":
	        ; // todo
	        
	        // "InstLPMLV2022_UnitModeStateManager".SC := TRUE; // Set state complete signal when action is done
	        
	      "LPMLV2022_STATE_SUSPENDED":
	        ; // todo
	        
	      "LPMLV2022_STATE_UNSUSPENDING":
	        ; // todo
	        
	        // "InstLPMLV2022_UnitModeStateManager".SC := TRUE; // Set state complete signal when action is done
	        
	      "LPMLV2022_STATE_COMPLETING":
	        ; // todo
	        
	        // "InstLPMLV2022_UnitModeStateManager".SC := TRUE; // Set state complete signal when action is done
	        
	      "LPMLV2022_STATE_COMPLETED":
	        ; // todo
	        
	      "LPMLV2022_STATE_ABORTING":
	        ; // todo
	        
	        // "InstLPMLV2022_UnitModeStateManager".SC := TRUE; // Set state complete signal when action is done
	        
	      "LPMLV2022_STATE_ABORTED":
	        ; // todo
	        
	      "LPMLV2022_STATE_CLEARING":
	        ; // todo
	        
	        // "InstLPMLV2022_UnitModeStateManager".SC := TRUE; // Set state complete signal when action is done
	        
	      ELSE
	        // Error reaction
	        ; // todo
	    END_CASE;
	  
	  "LPMLV2022_MODE_MANUAL":
	    CASE "InstLPMLV2022_UnitModeStateManager".StateCurrent OF
	    "LPMLV2022_STATE_RESETTING":
	      ; // todo
	      
	      // "InstLPMLV2022_UnitModeStateManager".SC := TRUE; // Set state complete signal when action is done
	      
	    "LPMLV2022_STATE_IDLE":
	      ; // todo
	      
	    "LPMLV2022_STATE_STARTING":
	      ; // todo
	      
	      // "InstLPMLV2022_UnitModeStateManager".SC := TRUE; // Set state complete signal when action is done
	      
	    "LPMLV2022_STATE_EXECUTE":
	      ; // todo
	      
	    "LPMLV2022_STATE_STOPPING":
	      ; // todo
	      
	      // "InstLPMLV2022_UnitModeStateManager".SC := TRUE; // Set state complete signal when action is done
	      
	    "LPMLV2022_STATE_STOPPED":
	      ; // todo
	      
	    "LPMLV2022_STATE_HOLDING":
	      ; // todo
	      
	      // "InstLPMLV2022_UnitModeStateManager".SC := TRUE; // Set state complete signal when action is done            
	      
	    "LPMLV2022_STATE_HELD":
	      ; // todo
	      
	    "LPMLV2022_STATE_UNHOLDING":
	      ; // todo
	      
	      // "InstLPMLV2022_UnitModeStateManager".SC := TRUE; // Set state complete signal when action is done   
	      
	    "LPMLV2022_STATE_SUSPENDING":
	      ; // todo
	      
	      // "InstLPMLV2022_UnitModeStateManager".SC := TRUE; // Set state complete signal when action is done
	      
	    "LPMLV2022_STATE_SUSPENDED":
	      ; // todo
	      
	    "LPMLV2022_STATE_UNSUSPENDING":
	      ; // todo
	      
	      // "InstLPMLV2022_UnitModeStateManager".SC := TRUE; // Set state complete signal when action is done
	      
	    "LPMLV2022_STATE_COMPLETING":
	      ; // todo
	      
	      // "InstLPMLV2022_UnitModeStateManager".SC := TRUE; // Set state complete signal when action is done
	      
	    "LPMLV2022_STATE_COMPLETED":
	      ; // todo
	      
	    "LPMLV2022_STATE_ABORTING":
	      ; // todo
	      
	      // "InstLPMLV2022_UnitModeStateManager".SC := TRUE; // Set state complete signal when action is done
	      
	    "LPMLV2022_STATE_ABORTED":
	      ; // todo
	      
	    "LPMLV2022_STATE_CLEARING":
	      ; // todo
	      
	      // "InstLPMLV2022_UnitModeStateManager".SC := TRUE; // Set state complete signal when action is done
	      
	    ELSE
	      // Error reaction
	      ; // todo
	  END_CASE;
	  
	  "LPMLV2022_MODE_USER_01":
	    CASE "InstLPMLV2022_UnitModeStateManager".StateCurrent OF
	      "LPMLV2022_STATE_RESETTING":
	        ; // todo
	        
	        // "InstLPMLV2022_UnitModeStateManager".SC := TRUE; // Set state complete signal when action is done
	        
	      "LPMLV2022_STATE_IDLE":
	        ; // todo
	        
	      "LPMLV2022_STATE_STARTING":
	        ; // todo
	        
	        // "InstLPMLV2022_UnitModeStateManager".SC := TRUE; // Set state complete signal when action is done
	        
	      "LPMLV2022_STATE_EXECUTE":
	        ; // todo
	        
	      "LPMLV2022_STATE_STOPPING":
	        ; // todo
	        
	        // "InstLPMLV2022_UnitModeStateManager".SC := TRUE; // Set state complete signal when action is done
	        
	      "LPMLV2022_STATE_STOPPED":
	        ; // todo
	        
	      "LPMLV2022_STATE_HOLDING":
	        ; // todo
	        
	        // "InstLPMLV2022_UnitModeStateManager".SC := TRUE; // Set state complete signal when action is done            
	        
	      "LPMLV2022_STATE_HELD":
	        ; // todo
	        
	      "LPMLV2022_STATE_UNHOLDING":
	        ; // todo
	        
	        // "InstLPMLV2022_UnitModeStateManager".SC := TRUE; // Set state complete signal when action is done   
	        
	      "LPMLV2022_STATE_SUSPENDING":
	        ; // todo
	        
	        // "InstLPMLV2022_UnitModeStateManager".SC := TRUE; // Set state complete signal when action is done
	        
	      "LPMLV2022_STATE_SUSPENDED":
	        ; // todo
	        
	      "LPMLV2022_STATE_UNSUSPENDING":
	        ; // todo
	        
	        // "InstLPMLV2022_UnitModeStateManager".SC := TRUE; // Set state complete signal when action is done
	        
	      "LPMLV2022_STATE_COMPLETING":
	        ; // todo
	        
	        // "InstLPMLV2022_UnitModeStateManager".SC := TRUE; // Set state complete signal when action is done
	        
	      "LPMLV2022_STATE_COMPLETED":
	        ; // todo
	        
	      "LPMLV2022_STATE_ABORTING":
	        ; // todo
	        
	        // "InstLPMLV2022_UnitModeStateManager".SC := TRUE; // Set state complete signal when action is done
	        
	      "LPMLV2022_STATE_ABORTED":
	        ; // todo
	        
	      "LPMLV2022_STATE_CLEARING":
	        ; // todo
	        
	        // "InstLPMLV2022_UnitModeStateManager".SC := TRUE; // Set state complete signal when action is done
	        
	      ELSE
	        // Error reaction
	        ; // todo
	    END_CASE;
	  
	  // "LPMLV2022_MODE_USER_02":
	  //   CASE "InstLPMLV2022_UnitModeStateManager".StateCurrent OF
	  //     "LPMLV2022_STATE_RESETTING":
	  //       ; // todo
	  
	  //       // "InstLPMLV2022_UnitModeStateManager".SC := TRUE; // Set state complete signal when action is done
	  
	  //     "LPMLV2022_STATE_IDLE":
	  //       ; // todo
	  
	  //     "LPMLV2022_STATE_STARTING":
	  //       ; // todo
	  
	  //       // "InstLPMLV2022_UnitModeStateManager".SC := TRUE; // Set state complete signal when action is done
	  
	  //     "LPMLV2022_STATE_EXECUTE":
	  //       ; // todo
	  
	  //     "LPMLV2022_STATE_STOPPING":
	  //       ; // todo
	  
	  //       // "InstLPMLV2022_UnitModeStateManager".SC := TRUE; // Set state complete signal when action is done
	  
	  //     "LPMLV2022_STATE_STOPPED":
	  //       ; // todo
	  
	  //     "LPMLV2022_STATE_HOLDING":
	  //       ; // todo
	  
	  //       // "InstLPMLV2022_UnitModeStateManager".SC := TRUE; // Set state complete signal when action is done            
	  
	  //     "LPMLV2022_STATE_HELD":
	  //       ; // todo
	  
	  //     "LPMLV2022_STATE_UNHOLDING":
	  //       ; // todo
	  
	  //       // "InstLPMLV2022_UnitModeStateManager".SC := TRUE; // Set state complete signal when action is done   
	  
	  //     "LPMLV2022_STATE_SUSPENDING":
	  //       ; // todo
	  
	  //       // "InstLPMLV2022_UnitModeStateManager".SC := TRUE; // Set state complete signal when action is done
	  
	  //     "LPMLV2022_STATE_SUSPENDED":
	  //       ; // todo
	  
	  //     "LPMLV2022_STATE_UNSUSPENDING":
	  //       ; // todo
	  
	  //       // "InstLPMLV2022_UnitModeStateManager".SC := TRUE; // Set state complete signal when action is done
	  
	  //     "LPMLV2022_STATE_COMPLETING":
	  //       ; // todo
	  
	  //       // "InstLPMLV2022_UnitModeStateManager".SC := TRUE; // Set state complete signal when action is done
	  
	  //     "LPMLV2022_STATE_COMPLETED":
	  //       ; // todo
	  
	  //     "LPMLV2022_STATE_ABORTING":
	  //       ; // todo
	  
	  //       // "InstLPMLV2022_UnitModeStateManager".SC := TRUE; // Set state complete signal when action is done
	  
	  //     "LPMLV2022_STATE_ABORTED":
	  //       ; // todo
	  
	  //     "LPMLV2022_STATE_CLEARING":
	  //       ; // todo
	  
	  //       // "InstLPMLV2022_UnitModeStateManager".SC := TRUE; // Set state complete signal when action is done
	  
	  //     ELSE
	  //       // Error reaction
	  //       ; // todo
	  //   END_CASE;
	
	ELSE
	  // Error reaction
	  ; // todo
	END_CASE;
END_FUNCTION_BLOCK

FUNCTION "LPMLV2022_ConfigureEnabledModesCfg" : Void
TITLE = LPMLV2022_ConfigureEnabledModesCfg
{ S7_Optimized_Access := 'TRUE' }
AUTHOR : APC_ERLF
FAMILY : OMAC
VERSION : 1.0
//Support: tech.team.motioncontrol@siemens.com
   VAR_INPUT 
      ProductionMode : Bool;   // TRUE: Enable unit mode Production
      MaintenanceMode : Bool;   // TRUE: Enable unit mode Maintenance
      UserMode01 : Bool;   // TRUE: Enable user-defined unit mode 01
      UserMode02 : Bool;   // TRUE: Enable user-defined unit mode 02
      UserMode03 : Bool;   // TRUE: Enable user-defined unit mode 03
      UserMode04 : Bool;   // TRUE: Enable user-defined unit mode 04
      UserMode05 : Bool;   // TRUE: Enable user-defined unit mode 05
      UserMode06 : Bool;   // TRUE: Enable user-defined unit mode 06
      UserMode07 : Bool;   // TRUE: Enable user-defined unit mode 07
      UserMode08 : Bool;   // TRUE: Enable user-defined unit mode 08
      UserMode09 : Bool;   // TRUE: Enable user-defined unit mode 09
      UserMode10 : Bool;   // TRUE: Enable user-defined unit mode 10
      UserMode11 : Bool;   // TRUE: Enable user-defined unit mode 11
      UserMode12 : Bool;   // TRUE: Enable user-defined unit mode 12
      UserMode13 : Bool;   // TRUE: Enable user-defined unit mode 13
      UserMode14 : Bool;   // TRUE: Enable user-defined unit mode 14
      UserMode15 : Bool;   // TRUE: Enable user-defined unit mode 15
      UserMode16 : Bool;   // TRUE: Enable user-defined unit mode 16
      UserMode17 : Bool;   // TRUE: Enable user-defined unit mode 17
      UserMode18 : Bool;   // TRUE: Enable user-defined unit mode 18
      UserMode19 : Bool;   // TRUE: Enable user-defined unit mode 19
      UserMode20 : Bool;   // TRUE: Enable user-defined unit mode 20
      UserMode21 : Bool;   // TRUE: Enable user-defined unit mode 21
      UserMode22 : Bool;   // TRUE: Enable user-defined unit mode 22
      UserMode23 : Bool;   // TRUE: Enable user-defined unit mode 23
      UserMode24 : Bool;   // TRUE: Enable user-defined unit mode 24
      UserMode25 : Bool;   // TRUE: Enable user-defined unit mode 25
      UserMode26 : Bool;   // TRUE: Enable user-defined unit mode 26
      UserMode27 : Bool;   // TRUE: Enable user-defined unit mode 27
      UserMode28 : Bool;   // TRUE: Enable user-defined unit mode 28
   END_VAR

   VAR_OUTPUT 
      EnabledModesCfg : DWord;   // Enabled unit modes configuration
   END_VAR


BEGIN
	REGION HEADER
	  //================================================================================
	  // SIEMENS AG
	  // (c)Copyright 2023 All Rights Reserved
	  //--------------------------------------------------------------------------------
	  // Library: LPMLV2022 
	  // Tested with: S7-1211 with FW version V4.2, S7-1511-1 PN with FW version V2.6
	  // Engineering: TIA Portal V15.1
	  // Restrictions: -
	  // Requirements: S7-1200 FW 4.2 / S7-1500 FW 2.6
	  // Functionality: The function generates the unit mode configuration as DWord.
	  // Support: tech.team.motioncontrol@siemens.com
	  // Note: Parameter comments are only available in language 'English (United States)'
	  //--------------------------------------------------------------------------------
	  // Change log table:
	  // Version  Date        Expert in charge  Changes applied
	  // 01.00.00 28.02.2023  KT                First released version
	  //================================================================================
	END_REGION
	
	// Initialize unitMode configuration
	#EnabledModesCfg := 16#0000_0008; // Note: mode Manual (EnabledModesCfg.%X3) is mandatory
	
	// Set unitMode configuration
	#EnabledModesCfg.%X1  := #ProductionMode;
	#EnabledModesCfg.%X2  := #MaintenanceMode;
	#EnabledModesCfg.%X4  := #UserMode01;
	#EnabledModesCfg.%X5  := #UserMode02;
	#EnabledModesCfg.%X6  := #UserMode03;
	#EnabledModesCfg.%X7  := #UserMode04;
	#EnabledModesCfg.%X8  := #UserMode05;
	#EnabledModesCfg.%X9  := #UserMode06;
	#EnabledModesCfg.%X10 := #UserMode07;
	#EnabledModesCfg.%X11 := #UserMode08;
	#EnabledModesCfg.%X12 := #UserMode09;
	#EnabledModesCfg.%X13 := #UserMode10;
	#EnabledModesCfg.%X14 := #UserMode11;
	#EnabledModesCfg.%X15 := #UserMode12;
	#EnabledModesCfg.%X16 := #UserMode13;
	#EnabledModesCfg.%X17 := #UserMode14;
	#EnabledModesCfg.%X18 := #UserMode15;
	#EnabledModesCfg.%X19 := #UserMode16;
	#EnabledModesCfg.%X20 := #UserMode17;
	#EnabledModesCfg.%X21 := #UserMode18;
	#EnabledModesCfg.%X22 := #UserMode19;
	#EnabledModesCfg.%X23 := #UserMode20;
	#EnabledModesCfg.%X24 := #UserMode21;
	#EnabledModesCfg.%X25 := #UserMode22;
	#EnabledModesCfg.%X26 := #UserMode23;
	#EnabledModesCfg.%X27 := #UserMode24;
	#EnabledModesCfg.%X28 := #UserMode25;
	#EnabledModesCfg.%X29 := #UserMode26;
	#EnabledModesCfg.%X30 := #UserMode27;
	#EnabledModesCfg.%X31 := #UserMode28;
END_FUNCTION

FUNCTION_BLOCK "ShowUnitModeStateManagerDiagnosticsInHMI"
{ S7_Optimized_Access := 'TRUE' }
VERSION : 0.1
   VAR_TEMP 
      tempDiagnosticsBufferIndexForHMI : Int;
      tempActualBufferIndex : Int;
   END_VAR


BEGIN
	REGION HEADER
	  //================================================================================
	  // SIEMENS AG
	  // (c)Copyright 2023 All Rights Reserved
	  //--------------------------------------------------------------------------------
	  // Library: -
	  // Tested with: S7-1513-1 PN with FW version V2.9
	  // Engineering: TIA Portal V17 Update 4
	  // Restrictions: -
	  // Requirements: LPMLV2022
	  // Functionality: Copies one element of diagnostics buffer for easier HMI access
	  // Support: tech.team.motioncontrol@siemens.com
	  // Note: Parameter comments are only available in language 'English (United States)'
	  //--------------------------------------------------------------------------------
	  // Change log table:
	  // Version  Date        Expert in charge  Changes applied
	  // 01.00.00 28.02.2023  KT                First released version
	  //================================================================================
	END_REGION
	
	// Create process image and verify the value for the index for selecting the diagnostics buffer entry to be displayed on the HMI
	#tempDiagnosticsBufferIndexForHMI := "UnitModeStateManagerDiagnosticsForHMI".diagnosticsBufferIndexForHMI;
	IF (#tempDiagnosticsBufferIndexForHMI < 0) THEN
	  #tempDiagnosticsBufferIndexForHMI := "LPMLV2022_DIAG_BUFFER_UPPER_LIM";
	  
	ELSIF (#tempDiagnosticsBufferIndexForHMI > "LPMLV2022_DIAG_BUFFER_UPPER_LIM") THEN
	  #tempDiagnosticsBufferIndexForHMI := 0;
	END_IF;
	
	// Copy the needed array element for HMI
	"UnitModeStateManagerDiagnosticsForHMI".diagnosticsBufferEntryForHMI := "InstLPMLV2022_UnitModeStateManager".diagnostics.buffer[#tempDiagnosticsBufferIndexForHMI];
	"UnitModeStateManagerDiagnosticsForHMI".diagnosticsBufferIndexForHMI := #tempDiagnosticsBufferIndexForHMI;
	
	// Provide actual diagnostics buffer index for HMI
	#tempActualBufferIndex := "InstLPMLV2022_UnitModeStateManager".diagnostics.bufferIndex;
	"UnitModeStateManagerDiagnosticsForHMI".actualDiagnosticsBufferIndex := #tempActualBufferIndex;
	
	// Provide actual diagnostics message for the HMI
	IF (#tempActualBufferIndex < 0) OR (#tempActualBufferIndex > "LPMLV2022_DIAG_BUFFER_UPPER_LIM") THEN // tempActualBufferIndex is invalid
	  "UnitModeStateManagerDiagnosticsForHMI".messageCurrentPLCIndex := 16#00;
	  
	ELSE // tempActualBufferIndex is valid, show corresponding message
	  "UnitModeStateManagerDiagnosticsForHMI".messageCurrentPLCIndex := "InstLPMLV2022_UnitModeStateManager".diagnostics.buffer[#tempActualBufferIndex].message;
	END_IF;
END_FUNCTION_BLOCK

FUNCTION_BLOCK "PACKMLV2022_PackTagsGlueCode"
{ S7_Optimized_Access := 'TRUE' }
VERSION : 0.1
   VAR_TEMP 
      tempUnitModeCurrent : DInt;   // Current Unit Mode Number (0: Invalid, 1: Production, 2: Maintenance, 3: Manual, 04 - 31: User Definable)
      tempStateCurrent : DInt;   // Current State Number (0: Undefined, 1: CLEARING, 2: STOPPED, 3: STARTING, 4: IDLE, 5: SUSPENDED, 6: EXECUTE, 7: STOPPING, 8: ABORTING, 9: ABORTED; 10: HOLDING, 11: HELD, 12: UNHOLDING, 13: SUSPENDING, 14: UNSUSPENDING, 15: RESETTING, 16: COMPLETING, 17: COMPLETED)
      tempReturnValue : Int;   // Return value from RD_LOC_T system function
      tempPLCDateTimeDTL {InstructionName := 'DTL'; LibVersion := '1.0'} : DTL;   // Current local time from the CPU clock (output from RD_LOC_T system function)
   END_VAR


BEGIN
	REGION COMMAND_TAGS
	  "InstLPMLV2022_UnitModeStateManager".UnitMode              := "PACKMLV2022".Command.UnitMode;
	  "InstLPMLV2022_UnitModeStateManager".UnitModeChangeRequest := "PACKMLV2022".Command.UnitModeChangeRequest;
	  
	  "InstLPMLV2022_UnitModeStateManager".CntrlCmd         := "PACKMLV2022".Command.CntrlCmd;
	  "InstLPMLV2022_UnitModeStateManager".CmdChangeRequest := "PACKMLV2022".Command.CmdChangeRequest;
	END_REGION
	
	#tempUnitModeCurrent := "InstLPMLV2022_UnitModeStateManager".UnitModeCurrent;
	#tempStateCurrent    := "InstLPMLV2022_UnitModeStateManager".StateCurrent;
	
	REGION STATUS_TAGS
	  "PACKMLV2022".Status.UnitModeCurrent := #tempUnitModeCurrent;
	  "PACKMLV2022".Status.StateCurrent    := #tempStateCurrent;
	  
	  "PACKMLV2022".Status.StateRequested       := "InstLPMLV2022_UnitModeStateManager".StateRequested;
	  "PACKMLV2022".Status.StateChangeInProcess := "InstLPMLV2022_UnitModeStateManager".StateChangeInProcess;
	  
	  // Call of LPMLV2022_Stacklight (OPTIONAL)
	  "InstLPMLV2022_Stacklight"(StateCurrent := #tempStateCurrent,
	                             Stacklight => "PACKMLV2022".Status.Stacklight[0]);
	END_REGION
	
	REGION ADMIN_TAGS
	  // Call of LPMLV2022_UnitModeStateTimes (OPTIONAL)
	  "InstLPMLV2022_UnitModeStateTimes"(UnitModeCurrent := #tempUnitModeCurrent,
	                                     StateCurrent := #tempStateCurrent);
	  
	  "PACKMLV2022".Admin.ModeTimeCurrent  := "InstLPMLV2022_UnitModeStateTimes".ModeTimeCurrent;
	  "PACKMLV2022".Admin.StateTimeCurrent := "InstLPMLV2022_UnitModeStateTimes".StateTimeCurrent;
	  
	  "PACKMLV2022".Admin.CumulativeTimes[0].AccTimeSinceReset := "InstLPMLV2022_UnitModeStateTimes".AccTimeSinceReset;
	  
	  // "PACKMLV2022".Admin.CumulativeTimes[0].ModeStateTimes["LPMLV2022_MODE_INVALID"].Mode  := "InstLPMLV2022_UnitModeStateTimes".cumulativeTimeAllModes["LPMLV2022_MODE_INVALID"];
	  // "PACKMLV2022".Admin.CumulativeTimes[0].ModeStateTimes["LPMLV2022_MODE_INVALID"].State := "InstLPMLV2022_UnitModeStateTimes".cumulativeTimeAllStatesOfAllModes["LPMLV2022_MODE_INVALID"];
	  
	  "PACKMLV2022".Admin.CumulativeTimes[0].ModeStateTimes["LPMLV2022_MODE_PRODUCTION"].Mode  := "InstLPMLV2022_UnitModeStateTimes".cumulativeTimeAllModes["LPMLV2022_MODE_PRODUCTION"];
	  "PACKMLV2022".Admin.CumulativeTimes[0].ModeStateTimes["LPMLV2022_MODE_PRODUCTION"].State := "InstLPMLV2022_UnitModeStateTimes".cumulativeTimeAllStatesOfAllModes["LPMLV2022_MODE_PRODUCTION"];
	  
	  "PACKMLV2022".Admin.CumulativeTimes[0].ModeStateTimes["LPMLV2022_MODE_MAINTENANCE"].Mode  := "InstLPMLV2022_UnitModeStateTimes".cumulativeTimeAllModes["LPMLV2022_MODE_MAINTENANCE"];
	  "PACKMLV2022".Admin.CumulativeTimes[0].ModeStateTimes["LPMLV2022_MODE_MAINTENANCE"].State := "InstLPMLV2022_UnitModeStateTimes".cumulativeTimeAllStatesOfAllModes["LPMLV2022_MODE_MAINTENANCE"];
	  
	  "PACKMLV2022".Admin.CumulativeTimes[0].ModeStateTimes["LPMLV2022_MODE_MANUAL"].Mode  := "InstLPMLV2022_UnitModeStateTimes".cumulativeTimeAllModes["LPMLV2022_MODE_MANUAL"];
	  "PACKMLV2022".Admin.CumulativeTimes[0].ModeStateTimes["LPMLV2022_MODE_MANUAL"].State := "InstLPMLV2022_UnitModeStateTimes".cumulativeTimeAllStatesOfAllModes["LPMLV2022_MODE_MANUAL"];
	  
	  "PACKMLV2022".Admin.CumulativeTimes[0].ModeStateTimes["LPMLV2022_MODE_USER_01"].Mode  := "InstLPMLV2022_UnitModeStateTimes".cumulativeTimeAllModes["LPMLV2022_MODE_USER_01"];
	  "PACKMLV2022".Admin.CumulativeTimes[0].ModeStateTimes["LPMLV2022_MODE_USER_01"].State := "InstLPMLV2022_UnitModeStateTimes".cumulativeTimeAllStatesOfAllModes["LPMLV2022_MODE_USER_01"];
	  
	  // "PACKMLV2022".Admin.CumulativeTimes[0].ModeStateTimes["LPMLV2022_MODE_USER_02"].Mode  := "InstLPMLV2022_UnitModeStateTimes".cumulativeTimeAllModes["LPMLV2022_MODE_USER_02"];
	  // "PACKMLV2022".Admin.CumulativeTimes[0].ModeStateTimes["LPMLV2022_MODE_USER_02"].State := "InstLPMLV2022_UnitModeStateTimes".cumulativeTimeAllStatesOfAllModes["LPMLV2022_MODE_USER_02"];
	  
